QRS_NEXT_CUT()
PTP {E1 28616.968,E2 28616.968}
PTP {X 0,Y 607.867,A -85,B 0,C 180,E1 28616.968,E2 28616.968,E3 0,E4 0,E5 0,E6 0}
QRS_SPEED_INIT()
LIN {X 0,Y 607.867,Z 1084,A -85,B 0,C 180,E1 28616.968,E2 28616.968,E3 0,E4 0,E5 0,E6 0} C_VEL
LIN {X 0,Y 607.867,Z 590.149,A -85,B 0,C 180,E1 28616.968,E2 28616.968} C_VEL
LIN {X 0,Y 607.867,Z 582.07,A -85,B 0,C 180,E1 28616.968,E2 28616.968} C_VEL
LIN {X 0,Y 607.876,Z 580.07,A -85,B 0,C 180,E1 28616.78,E2 28616.78} C_VEL
LIN {X 0,Y 607.89,Z 580.076,A -85,B 0,C 180,E1 28613.483,E2 28613.483} C_VEL
LIN {X 0,Y 607.884,Z 580.069,A -85,B 0,C 180,E1 28610.437,E2 28610.437} C_VEL
LIN {X 0,Y 607.889,Z 580.074,A -85,B 0,C 180,E1 28607.17,E2 28607.17} C_VEL
LIN {X 0,Y 607.897,Z 580.069,A -85,B 0,C 180,E1 28604.057,E2 28604.057} C_VEL
LIN {X 0,Y 607.881,Z 580.073,A -85,B 0,C 180,E1 28600.758,E2 28600.758} C_VEL
LIN {X 0,Y 607.908,Z 580.069,A -85,B 0,C 180,E1 28597.67,E2 28597.67} C_VEL
LIN {X 0,Y 607.882,Z 580.073,A -85,B 0,C 180,E1 28594.472,E2 28594.472} C_VEL
LIN {X 0,Y 607.917,Z 580.068,A -85,B 0,C 180,E1 28591.405,E2 28591.405} C_VEL
LIN {X 0,Y 607.88,Z 580.072,A -85,B 0,C 180,E1 28588.13,E2 28588.13} C_VEL
LIN {X 0,Y 607.913,Z 580.071,A -85,B 0,C 180,E1 28584.993,E2 28584.993} C_VEL
LIN {X 0,Y 607.881,Z 580.072,A -85,B 0,C 180,E1 28581.834,E2 28581.834} C_VEL
LIN {X 0,Y 607.911,Z 580.072,A -85,B 0,C 180,E1 28578.734,E2 28578.734} C_VEL
LIN {X 0,Y 607.907,Z 580.227,A -85,B 0,C 180,E1 28576.36,E2 28576.36} C_VEL
LIN {X 0,Y 607.894,Z 606.241,A -85,B 0,C 180,E1 28573.564,E2 28573.564} C_VEL
LIN {X 0,Y 607.911,Z 636.019,A -85,B 0,C 180,E1 28570.459,E2 28570.459} C_VEL
LIN {X 0,Y 607.889,Z 666.862,A -85,B 0,C 180,E1 28567.309,E2 28567.309} C_VEL
LIN {X 0,Y 607.91,Z 698.053,A -85,B 0,C 180,E1 28564.176,E2 28564.176} C_VEL
LIN {X 0,Y 607.909,Z 709.953,A -85,B 0,C 180,E1 28563.027,E2 28563.027} C_VEL
LIN {X 0,Y 607.905,Z 821.643,A -85,B 0,C 180,E1 28561.66,E2 28561.66} C_VEL
LIN {X 0,Y 607.917,Z 836.088,A -85,B 0,C 180,E1 28561.314,E2 28561.314} C_VEL
LIN {X 0,Y 607.919,Z 850.913,A -85,B 0,C 180,E1 28560.764,E2 28560.764} C_VEL
LIN {X 0,Y 607.91,Z 863.899,A -85,B 0,C 180,E1 28560.101,E2 28560.101} C_VEL
LIN {X 0,Y 607.919,Z 876.772,A -85,B 0,C 180,E1 28559.241,E2 28559.241} C_VEL
LIN {X 0,Y 607.919,Z 886.967,A -85,B 0,C 180,E1 28558.366,E2 28558.366} C_VEL
LIN {X 0,Y 607.917,Z 896.549,A -85,B 0,C 180,E1 28557.357,E2 28557.357} C_VEL
LIN {X 0,Y 607.917,Z 905.81,A -85,B 0,C 180,E1 28556.1,E2 28556.1} C_VEL
LIN {X 0,Y 607.915,Z 913.073,A -85,B 0,C 180,E1 28554.783,E2 28554.783} C_VEL
LIN {X 0,Y 607.916,Z 918.363,A -85,B 0,C 180,E1 28553.455,E2 28553.455} C_VEL
LIN {X 0,Y 607.917,Z 922.064,A -85,B 0,C 180,E1 28552.024,E2 28552.024} C_VEL
LIN {X 0,Y 607.916,Z 923.86,A -85,B 0,C 180,E1 28550.507,E2 28550.507} C_VEL
LIN {X 0,Y 607.917,Z 923.652,A -85,B 0,C 180,E1 28549.105,E2 28549.105} C_VEL
LIN {X 0,Y 607.915,Z 921.709,A -85,B 0,C 180,E1 28547.715,E2 28547.715} C_VEL
LIN {X 0,Y 607.914,Z 917.979,A -85,B 0,C 180,E1 28546.335,E2 28546.335} C_VEL
LIN {X 0,Y 607.919,Z 912.759,A -85,B 0,C 180,E1 28545.062,E2 28545.062} C_VEL
LIN {X 0,Y 607.918,Z 905.726,A -85,B 0,C 180,E1 28543.797,E2 28543.797} C_VEL
LIN {X 0,Y 607.919,Z 896.434,A -85,B 0,C 180,E1 28542.539,E2 28542.539} C_VEL
LIN {X 0,Y 607.917,Z 886.306,A -85,B 0,C 180,E1 28541.479,E2 28541.479} C_VEL
LIN {X 0,Y 607.916,Z 873.406,A -85,B 0,C 180,E1 28540.423,E2 28540.423} C_VEL
LIN {X 0,Y 607.898,Z 861.256,A -85,B 0,C 180,E1 28539.658,E2 28539.658} C_VEL
LIN {X 0,Y 607.918,Z 847.253,A -85,B 0,C 180,E1 28538.989,E2 28538.989} C_VEL
LIN {X 0,Y 607.919,Z 833.117,A -85,B 0,C 180,E1 28538.512,E2 28538.512} C_VEL
LIN {X 0,Y 607.905,Z 818.973,A -85,B 0,C 180,E1 28538.203,E2 28538.203} C_VEL
LIN {X 0,Y 607.918,Z 709.961,A -85,B 0,C 180,E1 28536.884,E2 28536.884} C_VEL
LIN {X 0,Y 607.915,Z 682.218,A -85,B 0,C 180,E1 28534.15,E2 28534.15} C_VEL
LIN {X 0,Y 607.91,Z 650.544,A -85,B 0,C 180,E1 28530.942,E2 28530.942} C_VEL
LIN {X 0,Y 607.909,Z 619.504,A -85,B 0,C 180,E1 28527.738,E2 28527.738} C_VEL
LIN {X 0,Y 607.919,Z 589.094,A -85,B 0,C 180,E1 28524.526,E2 28524.526} C_VEL
LIN {X 0,Y 607.905,Z 580.175,A -85,B 0,C 180,E1 28523.531,E2 28523.531} C_VEL
LIN {X 0,Y 607.898,Z 580.068,A -85,B 0,C 180,E1 28520.342,E2 28520.342} C_VEL
LIN {X 0,Y 607.902,Z 580.075,A -85,B 0,C 180,E1 28517.171,E2 28517.171} C_VEL
LIN {X 0,Y 607.895,Z 580.068,A -85,B 0,C 180,E1 28514.057,E2 28514.057} C_VEL
LIN {X 0,Y 607.903,Z 580.074,A -85,B 0,C 180,E1 28510.894,E2 28510.894} C_VEL
LIN {X 0,Y 607.892,Z 580.069,A -85,B 0,C 180,E1 28507.771,E2 28507.771} C_VEL
LIN {X 0,Y 607.904,Z 580.073,A -85,B 0,C 180,E1 28504.578,E2 28504.578} C_VEL
LIN {X 0,Y 607.888,Z 580.07,A -85,B 0,C 180,E1 28501.442,E2 28501.442} C_VEL
LIN {X 0,Y 607.906,Z 580.073,A -85,B 0,C 180,E1 28498.353,E2 28498.353} C_VEL
LIN {X 0,Y 607.886,Z 580.07,A -85,B 0,C 180,E1 28495.162,E2 28495.162} C_VEL
LIN {X 0,Y 607.905,Z 580.073,A -85,B 0,C 180,E1 28492.037,E2 28492.037} C_VEL
LIN {X 0,Y 607.886,Z 580.07,A -85,B 0,C 180,E1 28488.983,E2 28488.983} C_VEL
LIN {X 0,Y 607.906,Z 580.073,A -85,B 0,C 180,E1 28485.817,E2 28485.817} C_VEL
LIN {X 0,Y 607.882,Z 580.07,A -85,B 0,C 180,E1 28482.662,E2 28482.662} C_VEL
LIN {X 0,Y 607.908,Z 580.073,A -85,B 0,C 180,E1 28479.533,E2 28479.533} C_VEL
LIN {X 0,Y 607.88,Z 580.071,A -85,B 0,C 180,E1 28476.426,E2 28476.426} C_VEL
LIN {X 0,Y 607.912,Z 580.073,A -85,B 0,C 180,E1 28473.322,E2 28473.322} C_VEL
LIN {X 0,Y 607.879,Z 580.07,A -85,B 0,C 180,E1 28470.22,E2 28470.22} C_VEL
LIN {X 0,Y 607.914,Z 580.073,A -85,B 0,C 180,E1 28467.103,E2 28467.103} C_VEL
LIN {X 0,Y 607.877,Z 580.07,A -85,B 0,C 180,E1 28463.971,E2 28463.971} C_VEL
LIN {X 0,Y 607.916,Z 580.075,A -85,B 0,C 180,E1 28460.898,E2 28460.898} C_VEL
LIN {X 0,Y 607.876,Z 580.07,A -85,B 0,C 180,E1 28457.716,E2 28457.716} C_VEL
LIN {X 0,Y 607.917,Z 580.075,A -85,B 0,C 180,E1 28454.672,E2 28454.672} C_VEL
LIN {X 0,Y 607.875,Z 580.071,A -85,B 0,C 180,E1 28451.48,E2 28451.48} C_VEL
LIN {X 0,Y 607.918,Z 580.073,A -85,B 0,C 180,E1 28448.322,E2 28448.322} C_VEL
LIN {X 0,Y 607.871,Z 580.071,A -85,B 0,C 180,E1 28445.191,E2 28445.191} C_VEL
LIN {X 0,Y 607.917,Z 580.073,A -85,B 0,C 180,E1 28442.074,E2 28442.074} C_VEL
LIN {X 0,Y 607.868,Z 580.071,A -85,B 0,C 180,E1 28438.963,E2 28438.963} C_VEL
LIN {X 0,Y 607.918,Z 580.074,A -85,B 0,C 180,E1 28435.85,E2 28435.85} C_VEL
LIN {X 0,Y 607.866,Z 580.071,A -85,B 0,C 180,E1 28432.686,E2 28432.686} C_VEL
LIN {X 0,Y 607.919,Z 580.074,A -85,B 0,C 180,E1 28429.577,E2 28429.577} C_VEL
LIN {X 0,Y 607.864,Z 580.072,A -85,B 0,C 180,E1 28426.441,E2 28426.441} C_VEL
LIN {X 0,Y 607.918,Z 580.075,A -85,B 0,C 180,E1 28423.371,E2 28423.371} C_VEL
LIN {X 0,Y 607.863,Z 580.072,A -85,B 0,C 180,E1 28420.194,E2 28420.194} C_VEL
LIN {X 0,Y 607.914,Z 580.077,A -85,B 0,C 180,E1 28417.16,E2 28417.16} C_VEL
LIN {X 0,Y 607.867,Z 580.071,A -85,B 0,C 180,E1 28414.053,E2 28414.053} C_VEL
LIN {X 0,Y 607.913,Z 580.078,A -85,B 0,C 180,E1 28410.975,E2 28410.975} C_VEL
LIN {X 0,Y 607.864,Z 580.072,A -85,B 0,C 180,E1 28407.796,E2 28407.796} C_VEL
LIN {X 0,Y 607.906,Z 580.078,A -85,B 0,C 180,E1 28404.738,E2 28404.738} C_VEL
LIN {X 0,Y 607.862,Z 580.072,A -85,B 0,C 180,E1 28401.555,E2 28401.555} C_VEL
LIN {X 0,Y 607.894,Z 580.077,A -85,B 0,C 180,E1 28398.593,E2 28398.593} C_VEL
LIN {X 0,Y 607.867,Z 580.071,A -85,B 0,C 180,E1 28395.384,E2 28395.384} C_VEL
LIN {X 0,Y 607.886,Z 580.077,A -85,B 0,C 180,E1 28392.394,E2 28392.394} C_VEL
LIN {X 0,Y 607.869,Z 580.072,A -85,B 0,C 180,E1 28389.171,E2 28389.171} C_VEL
LIN {X 0,Y 607.869,Z 580.076,A -85,B 0,C 180,E1 28386.295,E2 28386.295} C_VEL
LIN {X 0,Y 607.889,Z 580.07,A -85,B 0,C 180,E1 28383.099,E2 28383.099} C_VEL
LIN {X 0,Y 607.865,Z 580.075,A -85,B 0,C 180,E1 28380.094,E2 28380.094} C_VEL
LIN {X 0,Y 607.896,Z 580.312,A -85,B 0,C 180,E1 28379.784,E2 28379.784} C_VEL
LIN {X 0,Y 607.918,Z 589.008,A -85,B 0,C 180,E1 28379.15,E2 28379.15} C_VEL
LIN {X 0,Y 607.866,Z 632.567,A -85,B 0,C 180,E1 28376.209,E2 28376.209} C_VEL
LIN {X 0,Y 607.91,Z 678.154,A -85,B 0,C 180,E1 28373.205,E2 28373.205} C_VEL
LIN {X 0,Y 607.897,Z 691.997,A -85,B 0,C 180,E1 28372.331,E2 28372.331} C_VEL
LIN {X 0,Y 607.914,Z 901.305,A -85,B 0,C 180,E1 28369.705,E2 28369.705} C_VEL
LIN {X 0,Y 607.901,Z 919.582,A -85,B 0,C 180,E1 28369.305,E2 28369.305} C_VEL
LIN {X 0,Y 607.918,Z 938.403,A -85,B 0,C 180,E1 28368.707,E2 28368.707} C_VEL
LIN {X 0,Y 607.886,Z 956.055,A -85,B 0,C 180,E1 28367.963,E2 28367.963} C_VEL
LIN {X 0,Y 607.919,Z 972.787,A -85,B 0,C 180,E1 28367.073,E2 28367.073} C_VEL
LIN {X 0,Y 607.916,Z 988.639,A -85,B 0,C 180,E1 28366.041,E2 28366.041} C_VEL
LIN {X 0,Y 607.918,Z 1003.56,A -85,B 0,C 180,E1 28364.867,E2 28364.867} C_VEL
LIN {X 0,Y 607.918,Z 1017.218,A -85,B 0,C 180,E1 28363.582,E2 28363.582} C_VEL
LIN {X 0,Y 607.916,Z 1029.905,A -85,B 0,C 180,E1 28362.153,E2 28362.153} C_VEL
LIN {X 0,Y 607.915,Z 1041.223,A -85,B 0,C 180,E1 28360.615,E2 28360.615} C_VEL
LIN {X 0,Y 607.918,Z 1050.988,A -85,B 0,C 180,E1 28358.989,E2 28358.989} C_VEL
LIN {X 0,Y 607.909,Z 1058.863,A -85,B 0,C 180,E1 28357.35,E2 28357.35} C_VEL
LIN {X 0,Y 607.906,Z 1065.107,A -85,B 0,C 180,E1 28355.664,E2 28355.664} C_VEL
LIN {X 0,Y 607.916,Z 1069.872,A -85,B 0,C 180,E1 28353.867,E2 28353.867} C_VEL
LIN {X 0,Y 607.916,Z 1072.787,A -85,B 0,C 180,E1 28352.074,E2 28352.074} C_VEL
LIN {X 0,Y 607.907,Z 1073.94,A -85,B 0,C 180,E1 28350.283,E2 28350.283} C_VEL
LIN {X 0,Y 607.915,Z 1073.348,A -85,B 0,C 180,E1 28348.492,E2 28348.492} C_VEL
LIN {X 0,Y 607.908,Z 1071.005,A -85,B 0,C 180,E1 28346.7,E2 28346.7} C_VEL
LIN {X 0,Y 607.905,Z 1067.096,A -85,B 0,C 180,E1 28344.999,E2 28344.999} C_VEL
LIN {X 0,Y 607.914,Z 1061.467,A -85,B 0,C 180,E1 28343.294,E2 28343.294} C_VEL
LIN {X 0,Y 607.918,Z 1054.423,A -85,B 0,C 180,E1 28341.678,E2 28341.678} C_VEL
LIN {X 0,Y 607.91,Z 1045.509,A -85,B 0,C 180,E1 28340.055,E2 28340.055} C_VEL
LIN {X 0,Y 607.919,Z 1035.145,A -85,B 0,C 180,E1 28338.521,E2 28338.521} C_VEL
LIN {X 0,Y 607.914,Z 1023.346,A -85,B 0,C 180,E1 28337.075,E2 28337.075} C_VEL
LIN {X 0,Y 607.915,Z 1010.089,A -85,B 0,C 180,E1 28335.717,E2 28335.717} C_VEL
LIN {X 0,Y 607.917,Z 995.234,A -85,B 0,C 180,E1 28334.449,E2 28334.449} C_VEL
LIN {X 0,Y 607.918,Z 979.217,A -85,B 0,C 180,E1 28333.321,E2 28333.321} C_VEL
LIN {X 0,Y 607.895,Z 963.025,A -85,B 0,C 180,E1 28332.384,E2 28332.384} C_VEL
LIN {X 0,Y 607.907,Z 946.062,A -85,B 0,C 180,E1 28331.591,E2 28331.591} C_VEL
LIN {X 0,Y 607.905,Z 927.374,A -85,B 0,C 180,E1 28330.92,E2 28330.92} C_VEL
LIN {X 0,Y 607.905,Z 909.317,A -85,B 0,C 180,E1 28330.449,E2 28330.449} C_VEL
LIN {X 0,Y 607.919,Z 889.788,A -85,B 0,C 180,E1 28330.128,E2 28330.128} C_VEL
LIN {X 0,Y 607.896,Z 691.355,A -85,B 0,C 180,E1 28327.646,E2 28327.646} C_VEL
LIN {X 0,Y 607.914,Z 645.175,A -85,B 0,C 180,E1 28324.631,E2 28324.631} C_VEL
LIN {X 0,Y 607.917,Z 598.704,A -85,B 0,C 180,E1 28321.512,E2 28321.512} C_VEL
LIN {X 0,Y 607.898,Z 580.397,A -85,B 0,C 180,E1 28320.232,E2 28320.232} C_VEL
LIN {X 0,Y 607.853,Z 580.073,A -85,B 0,C 180,E1 28319.342,E2 28319.342} C_VEL
LIN {X 0,Y 607.909,Z 580.078,A -85,B 0,C 180,E1 28316.16,E2 28316.16} C_VEL
LIN {X 0,Y 607.847,Z 580.075,A -85,B 0,C 180,E1 28313.22,E2 28313.22} C_VEL
LIN {X 0,Y 607.918,Z 580.073,A -85,B 0,C 180,E1 28310.182,E2 28310.182} C_VEL
LIN {X 0,Y 607.848,Z 580.075,A -85,B 0,C 180,E1 28307.192,E2 28307.192} C_VEL
LIN {X 0,Y 607.919,Z 580.069,A -85,B 0,C 180,E1 28304.184,E2 28304.184} C_VEL
LIN {X 0,Y 607.851,Z 580.076,A -85,B 0,C 180,E1 28301.02,E2 28301.02} C_VEL
LIN {X 0,Y 607.909,Z 580.069,A -85,B 0,C 180,E1 28298.016,E2 28298.016} C_VEL
LIN {X 0,Y 607.855,Z 580.076,A -85,B 0,C 180,E1 28294.835,E2 28294.835} C_VEL
LIN {X 0,Y 607.897,Z 580.069,A -85,B 0,C 180,E1 28291.869,E2 28291.869} C_VEL
LIN {X 0,Y 607.862,Z 580.076,A -85,B 0,C 180,E1 28288.705,E2 28288.705} C_VEL
LIN {X 0,Y 607.886,Z 580.07,A -85,B 0,C 180,E1 28285.736,E2 28285.736} C_VEL
LIN {X 0,Y 607.869,Z 580.077,A -85,B 0,C 180,E1 28282.535,E2 28282.535} C_VEL
LIN {X 0,Y 607.876,Z 580.07,A -85,B 0,C 180,E1 28279.606,E2 28279.606} C_VEL
LIN {X 0,Y 607.873,Z 580.077,A -85,B 0,C 180,E1 28276.336,E2 28276.336} C_VEL
LIN {X 0,Y 607.882,Z 580.07,A -85,B 0,C 180,E1 28273.313,E2 28273.313} C_VEL
LIN {X 0,Y 607.875,Z 580.076,A -85,B 0,C 180,E1 28270.041,E2 28270.041} C_VEL
LIN {X 0,Y 607.891,Z 580.069,A -85,B 0,C 180,E1 28266.991,E2 28266.991} C_VEL
LIN {X 0,Y 607.875,Z 580.076,A -85,B 0,C 180,E1 28263.772,E2 28263.772} C_VEL
LIN {X 0,Y 607.889,Z 580.069,A -85,B 0,C 180,E1 28260.754,E2 28260.754} C_VEL
LIN {X 0,Y 607.881,Z 580.075,A -85,B 0,C 180,E1 28257.549,E2 28257.549} C_VEL
LIN {X 0,Y 607.876,Z 580.07,A -85,B 0,C 180,E1 28256.78,E2 28256.78} C_VEL
LIN {X 0,Y 606.932,Z 580.196,A -85,B 0,C 180,E1 28256.054,E2 28256.054} C_VEL
LIN {X 0,Y 600.424,Z 581.012,A -85,B 0,C 180,E1 28253.964,E2 28253.964} C_VEL
LIN {X 0,Y 599.952,Z 581.065,A -85,B 0,C 180,E1 28253.487,E2 28253.487} C_VEL
LIN {X 0,Y 599.948,Z 581.058,A -85,B 0,C 180,E1 28250.406,E2 28250.406} C_VEL
LIN {X 0,Y 599.944,Z 581.063,A -85,B 0,C 180,E1 28247.096,E2 28247.096} C_VEL
LIN {X 0,Y 599.971,Z 581.057,A -85,B 0,C 180,E1 28243.94,E2 28243.94} C_VEL
LIN {X 0,Y 599.94,Z 581.062,A -85,B 0,C 180,E1 28240.732,E2 28240.732} C_VEL
LIN {X 0,Y 599.97,Z 581.058,A -85,B 0,C 180,E1 28237.656,E2 28237.656} C_VEL
LIN {X 0,Y 599.941,Z 581.062,A -85,B 0,C 180,E1 28234.427,E2 28234.427} C_VEL
LIN {X 0,Y 599.974,Z 581.059,A -85,B 0,C 180,E1 28231.317,E2 28231.317} C_VEL
LIN {X 0,Y 599.941,Z 581.061,A -85,B 0,C 180,E1 28228.108,E2 28228.108} C_VEL
LIN {X 0,Y 599.975,Z 581.059,A -85,B 0,C 180,E1 28225.021,E2 28225.021} C_VEL
LIN {X 0,Y 599.942,Z 581.061,A -85,B 0,C 180,E1 28221.807,E2 28221.807} C_VEL
LIN {X 0,Y 599.972,Z 581.062,A -85,B 0,C 180,E1 28218.704,E2 28218.704} C_VEL
LIN {X 0,Y 600.003,Z 581.296,A -85,B 0,C 180,E1 28216.611,E2 28216.611} C_VEL
LIN {X 0,Y 600.305,Z 585.322,A -85,B 0,C 180,E1 28216.141,E2 28216.141} C_VEL
LIN {X 0,Y 600.216,Z 615.031,A -85,B 0,C 180,E1 28212.947,E2 28212.947} C_VEL
LIN {X 0,Y 600.138,Z 645.674,A -85,B 0,C 180,E1 28209.729,E2 28209.729} C_VEL
LIN {X 0,Y 600.077,Z 677.028,A -85,B 0,C 180,E1 28206.501,E2 28206.501} C_VEL
LIN {X 0,Y 600.029,Z 709.286,A -85,B 0,C 180,E1 28203.246,E2 28203.246} C_VEL
LIN {X 0,Y 600.113,Z 712.197,A -85,B 0,C 180,E1 28203.155,E2 28203.155} C_VEL
LIN {X 0,Y 600.068,Z 821.391,A -85,B 0,C 180,E1 28201.819,E2 28201.819} C_VEL
LIN {X 0,Y 600.062,Z 836.233,A -85,B 0,C 180,E1 28201.461,E2 28201.461} C_VEL
LIN {X 0,Y 600.039,Z 850.43,A -85,B 0,C 180,E1 28200.929,E2 28200.929} C_VEL
LIN {X 0,Y 600.003,Z 863.74,A -85,B 0,C 180,E1 28200.246,E2 28200.246} C_VEL
LIN {X 0,Y 599.985,Z 876.43,A -85,B 0,C 180,E1 28199.392,E2 28199.392} C_VEL
LIN {X 0,Y 599.962,Z 887.649,A -85,B 0,C 180,E1 28198.411,E2 28198.411} C_VEL
LIN {X 0,Y 599.942,Z 897.114,A -85,B 0,C 180,E1 28197.386,E2 28197.386} C_VEL
LIN {X 0,Y 599.931,Z 905.633,A -85,B 0,C 180,E1 28196.21,E2 28196.21} C_VEL
LIN {X 0,Y 599.923,Z 912.634,A -85,B 0,C 180,E1 28194.939,E2 28194.939} C_VEL
LIN {X 0,Y 599.92,Z 917.785,A -85,B 0,C 180,E1 28193.682,E2 28193.682} C_VEL
LIN {X 0,Y 599.917,Z 921.699,A -85,B 0,C 180,E1 28192.23,E2 28192.23} C_VEL
LIN {X 0,Y 599.918,Z 923.597,A -85,B 0,C 180,E1 28190.895,E2 28190.895} C_VEL
LIN {X 0,Y 599.915,Z 923.894,A -85,B 0,C 180,E1 28189.471,E2 28189.471} C_VEL
LIN {X 0,Y 599.917,Z 922.396,A -85,B 0,C 180,E1 28188.059,E2 28188.059} C_VEL
LIN {X 0,Y 599.917,Z 919.149,A -85,B 0,C 180,E1 28186.658,E2 28186.658} C_VEL
LIN {X 0,Y 599.919,Z 914.02,A -85,B 0,C 180,E1 28185.268,E2 28185.268} C_VEL
LIN {X 0,Y 599.93,Z 907.355,A -85,B 0,C 180,E1 28183.984,E2 28183.984} C_VEL
LIN {X 0,Y 599.936,Z 899.376,A -85,B 0,C 180,E1 28182.806,E2 28182.806} C_VEL
LIN {X 0,Y 599.958,Z 889.975,A -85,B 0,C 180,E1 28181.731,E2 28181.731} C_VEL
LIN {X 0,Y 599.977,Z 880.494,A -85,B 0,C 180,E1 28180.854,E2 28180.854} C_VEL
LIN {X 0,Y 599.976,Z 869.55,A -85,B 0,C 180,E1 28180.029,E2 28180.029} C_VEL
LIN {X 0,Y 600.023,Z 857.202,A -85,B 0,C 180,E1 28179.302,E2 28179.302} C_VEL
LIN {X 0,Y 600.05,Z 842.832,A -85,B 0,C 180,E1 28178.673,E2 28178.673} C_VEL
LIN {X 0,Y 600.074,Z 828.414,A -85,B 0,C 180,E1 28178.238,E2 28178.238} C_VEL
LIN {X 0,Y 600.07,Z 813.09,A -85,B 0,C 180,E1 28177.966,E2 28177.966} C_VEL
LIN {X 0,Y 600.055,Z 710.005,A -85,B 0,C 180,E1 28176.711,E2 28176.711} C_VEL
LIN {X 0,Y 600.033,Z 688.618,A -85,B 0,C 180,E1 28174.588,E2 28174.588} C_VEL
LIN {X 0,Y 600.092,Z 657.766,A -85,B 0,C 180,E1 28171.432,E2 28171.432} C_VEL
LIN {X 0,Y 600.176,Z 627.511,A -85,B 0,C 180,E1 28168.281,E2 28168.281} C_VEL
LIN {X 0,Y 600.269,Z 597.858,A -85,B 0,C 180,E1 28165.127,E2 28165.127} C_VEL
LIN {X 0,Y 600.134,Z 582.003,A -85,B 0,C 180,E1 28163.399,E2 28163.399} C_VEL
LIN {X 0,Y 599.961,Z 581.085,A -85,B 0,C 180,E1 28163.204,E2 28163.204} C_VEL
LIN {X 0,Y 599.954,Z 581.061,A -85,B 0,C 180,E1 28160.045,E2 28160.045} C_VEL
LIN {X 0,Y 599.96,Z 581.06,A -85,B 0,C 180,E1 28156.9,E2 28156.9} C_VEL
LIN {X 0,Y 599.952,Z 581.061,A -85,B 0,C 180,E1 28153.741,E2 28153.741} C_VEL
LIN {X 0,Y 599.963,Z 581.058,A -85,B 0,C 180,E1 28150.53,E2 28150.53} C_VEL
LIN {X 0,Y 599.954,Z 581.062,A -85,B 0,C 180,E1 28147.357,E2 28147.357} C_VEL
LIN {X 0,Y 599.971,Z 581.056,A -85,B 0,C 180,E1 28144.111,E2 28144.111} C_VEL
LIN {X 0,Y 599.973,Z 581.065,A -85,B 0,C 180,E1 28140.772,E2 28140.772} C_VEL
LIN {X 0,Y 599.954,Z 581.056,A -85,B 0,C 180,E1 28137.432,E2 28137.432} C_VEL
LIN {X 0,Y 599.97,Z 581.063,A -85,B 0,C 180,E1 28134.252,E2 28134.252} C_VEL
LIN {X 0,Y 599.948,Z 581.058,A -85,B 0,C 180,E1 28131.075,E2 28131.075} C_VEL
LIN {X 0,Y 599.97,Z 581.062,A -85,B 0,C 180,E1 28127.937,E2 28127.937} C_VEL
LIN {X 0,Y 599.945,Z 581.059,A -85,B 0,C 180,E1 28124.767,E2 28124.767} C_VEL
LIN {X 0,Y 599.971,Z 581.061,A -85,B 0,C 180,E1 28121.678,E2 28121.678} C_VEL
LIN {X 0,Y 599.944,Z 581.059,A -85,B 0,C 180,E1 28118.558,E2 28118.558} C_VEL
LIN {X 0,Y 599.97,Z 581.062,A -85,B 0,C 180,E1 28115.419,E2 28115.419} C_VEL
LIN {X 0,Y 599.943,Z 581.058,A -85,B 0,C 180,E1 28112.331,E2 28112.331} C_VEL
LIN {X 0,Y 599.975,Z 581.062,A -85,B 0,C 180,E1 28109.161,E2 28109.161} C_VEL
LIN {X 0,Y 599.938,Z 581.058,A -85,B 0,C 180,E1 28105.997,E2 28105.997} C_VEL
LIN {X 0,Y 599.974,Z 581.062,A -85,B 0,C 180,E1 28102.849,E2 28102.849} C_VEL
LIN {X 0,Y 599.937,Z 581.06,A -85,B 0,C 180,E1 28099.775,E2 28099.775} C_VEL
LIN {X 0,Y 599.974,Z 581.061,A -85,B 0,C 180,E1 28096.615,E2 28096.615} C_VEL
LIN {X 0,Y 599.934,Z 581.06,A -85,B 0,C 180,E1 28093.493,E2 28093.493} C_VEL
LIN {X 0,Y 599.977,Z 581.06,A -85,B 0,C 180,E1 28090.369,E2 28090.369} C_VEL
LIN {X 0,Y 599.934,Z 581.059,A -85,B 0,C 180,E1 28087.277,E2 28087.277} C_VEL
LIN {X 0,Y 599.977,Z 581.062,A -85,B 0,C 180,E1 28084.11,E2 28084.11} C_VEL
LIN {X 0,Y 599.927,Z 581.06,A -85,B 0,C 180,E1 28080.955,E2 28080.955} C_VEL
LIN {X 0,Y 599.978,Z 581.063,A -85,B 0,C 180,E1 28077.899,E2 28077.899} C_VEL
LIN {X 0,Y 599.927,Z 581.061,A -85,B 0,C 180,E1 28074.741,E2 28074.741} C_VEL
LIN {X 0,Y 599.979,Z 581.063,A -85,B 0,C 180,E1 28071.664,E2 28071.664} C_VEL
LIN {X 0,Y 599.926,Z 581.061,A -85,B 0,C 180,E1 28068.519,E2 28068.519} C_VEL
LIN {X 0,Y 599.98,Z 581.063,A -85,B 0,C 180,E1 28065.426,E2 28065.426} C_VEL
LIN {X 0,Y 599.928,Z 581.061,A -85,B 0,C 180,E1 28062.343,E2 28062.343} C_VEL
LIN {X 0,Y 599.978,Z 581.064,A -85,B 0,C 180,E1 28059.214,E2 28059.214} C_VEL
LIN {X 0,Y 599.927,Z 581.061,A -85,B 0,C 180,E1 28056.11,E2 28056.11} C_VEL
LIN {X 0,Y 599.977,Z 581.065,A -85,B 0,C 180,E1 28053.045,E2 28053.045} C_VEL
LIN {X 0,Y 599.926,Z 581.06,A -85,B 0,C 180,E1 28049.882,E2 28049.882} C_VEL
LIN {X 0,Y 599.966,Z 581.066,A -85,B 0,C 180,E1 28046.865,E2 28046.865} C_VEL
LIN {X 0,Y 599.932,Z 581.06,A -85,B 0,C 180,E1 28043.726,E2 28043.726} C_VEL
LIN {X 0,Y 599.951,Z 581.065,A -85,B 0,C 180,E1 28040.706,E2 28040.706} C_VEL
LIN {X 0,Y 599.925,Z 581.061,A -85,B 0,C 180,E1 28037.417,E2 28037.417} C_VEL
LIN {X 0,Y 599.963,Z 581.066,A -85,B 0,C 180,E1 28034.362,E2 28034.362} C_VEL
LIN {X 0,Y 599.92,Z 581.062,A -85,B 0,C 180,E1 28031.121,E2 28031.121} C_VEL
LIN {X 0,Y 599.966,Z 581.066,A -85,B 0,C 180,E1 28028.07,E2 28028.07} C_VEL
LIN {X 0,Y 599.919,Z 581.063,A -85,B 0,C 180,E1 28024.867,E2 28024.867} C_VEL
LIN {X 0,Y 599.955,Z 581.066,A -85,B 0,C 180,E1 28021.891,E2 28021.891} C_VEL
LIN {X 0,Y 599.958,Z 581.314,A -85,B 0,C 180,E1 28020.144,E2 28020.144} C_VEL
LIN {X 0,Y 600.654,Z 584.52,A -85,B 0,C 180,E1 28019.85,E2 28019.85} C_VEL
LIN {X 0,Y 600.468,Z 627.841,A -85,B 0,C 180,E1 28016.878,E2 28016.878} C_VEL
LIN {X 0,Y 600.389,Z 672.736,A -85,B 0,C 180,E1 28013.871,E2 28013.871} C_VEL
LIN {X 0,Y 600.409,Z 692.171,A -85,B 0,C 180,E1 28012.621,E2 28012.621} C_VEL
LIN {X 0,Y 600.373,Z 901.305,A -85,B 0,C 180,E1 28009.963,E2 28009.963} C_VEL
LIN {X 0,Y 600.32,Z 920.323,A -85,B 0,C 180,E1 28009.538,E2 28009.538} C_VEL
LIN {X 0,Y 600.29,Z 938.402,A -85,B 0,C 180,E1 28008.954,E2 28008.954} C_VEL
LIN {X 0,Y 600.204,Z 956.053,A -85,B 0,C 180,E1 28008.201,E2 28008.201} C_VEL
LIN {X 0,Y 600.18,Z 972.703,A -85,B 0,C 180,E1 28007.305,E2 28007.305} C_VEL
LIN {X 0,Y 600.122,Z 988.638,A -85,B 0,C 180,E1 28006.255,E2 28006.255} C_VEL
LIN {X 0,Y 600.069,Z 1003.561,A -85,B 0,C 180,E1 28005.066,E2 28005.066} C_VEL
LIN {X 0,Y 600.02,Z 1017.017,A -85,B 0,C 180,E1 28003.786,E2 28003.786} C_VEL
LIN {X 0,Y 599.983,Z 1029.906,A -85,B 0,C 180,E1 28002.317,E2 28002.317} C_VEL
LIN {X 0,Y 599.956,Z 1041.224,A -85,B 0,C 180,E1 28000.758,E2 28000.758} C_VEL
LIN {X 0,Y 599.934,Z 1050.989,A -85,B 0,C 180,E1 27999.11,E2 27999.11} C_VEL
LIN {X 0,Y 599.92,Z 1059.042,A -85,B 0,C 180,E1 27997.406,E2 27997.406} C_VEL
LIN {X 0,Y 599.91,Z 1065.409,A -85,B 0,C 180,E1 27995.643,E2 27995.643} C_VEL
LIN {X 0,Y 599.916,Z 1069.873,A -85,B 0,C 180,E1 27993.918,E2 27993.918} C_VEL
LIN {X 0,Y 599.917,Z 1072.787,A -85,B 0,C 180,E1 27992.102,E2 27992.102} C_VEL
LIN {X 0,Y 599.907,Z 1073.94,A -85,B 0,C 180,E1 27990.287,E2 27990.287} C_VEL
LIN {X 0,Y 599.915,Z 1073.348,A -85,B 0,C 180,E1 27988.472,E2 27988.472} C_VEL
LIN {X 0,Y 599.907,Z 1071.005,A -85,B 0,C 180,E1 27986.656,E2 27986.656} C_VEL
LIN {X 0,Y 599.908,Z 1067.097,A -85,B 0,C 180,E1 27984.932,E2 27984.932} C_VEL
LIN {X 0,Y 599.92,Z 1061.468,A -85,B 0,C 180,E1 27983.204,E2 27983.204} C_VEL
LIN {X 0,Y 599.931,Z 1054.423,A -85,B 0,C 180,E1 27981.567,E2 27981.567} C_VEL
LIN {X 0,Y 599.942,Z 1045.51,A -85,B 0,C 180,E1 27979.922,E2 27979.922} C_VEL
LIN {X 0,Y 599.969,Z 1035.146,A -85,B 0,C 180,E1 27978.367,E2 27978.367} C_VEL
LIN {X 0,Y 600,Z 1023.346,A -85,B 0,C 180,E1 27976.901,E2 27976.901} C_VEL
LIN {X 0,Y 600.047,Z 1009.759,A -85,B 0,C 180,E1 27975.494,E2 27975.494} C_VEL
LIN {X 0,Y 600.103,Z 995.233,A -85,B 0,C 180,E1 27974.242,E2 27974.242} C_VEL
LIN {X 0,Y 600.165,Z 979.22,A -85,B 0,C 180,E1 27973.099,E2 27973.099} C_VEL
LIN {X 0,Y 600.195,Z 962.033,A -85,B 0,C 180,E1 27972.1,E2 27972.1} C_VEL
LIN {X 0,Y 600.277,Z 944.644,A -85,B 0,C 180,E1 27971.293,E2 27971.293} C_VEL
LIN {X 0,Y 600.315,Z 926.513,A -85,B 0,C 180,E1 27970.644,E2 27970.644} C_VEL
LIN {X 0,Y 600.358,Z 908.143,A -85,B 0,C 180,E1 27970.17,E2 27970.17} C_VEL
LIN {X 0,Y 600.395,Z 888.268,A -85,B 0,C 180,E1 27969.85,E2 27969.85} C_VEL
LIN {X 0,Y 600.37,Z 691.85,A -85,B 0,C 180,E1 27967.371,E2 27967.371} C_VEL
LIN {X 0,Y 600.463,Z 645.962,A -85,B 0,C 180,E1 27964.346,E2 27964.346} C_VEL
LIN {X 0,Y 600.604,Z 599.492,A -85,B 0,C 180,E1 27961.187,E2 27961.187} C_VEL
LIN {X 0,Y 600.562,Z 583.327,A -85,B 0,C 180,E1 27960.062,E2 27960.062} C_VEL
LIN {X 0,Y 599.949,Z 581.259,A -85,B 0,C 180,E1 27959.842,E2 27959.842} C_VEL
LIN {X 0,Y 599.943,Z 581.06,A -85,B 0,C 180,E1 27956.96,E2 27956.96} C_VEL
LIN {X 0,Y 599.93,Z 581.066,A -85,B 0,C 180,E1 27953.726,E2 27953.726} C_VEL
LIN {X 0,Y 599.933,Z 581.061,A -85,B 0,C 180,E1 27950.803,E2 27950.803} C_VEL
LIN {X 0,Y 599.936,Z 581.066,A -85,B 0,C 180,E1 27947.548,E2 27947.548} C_VEL
LIN {X 0,Y 599.934,Z 581.06,A -85,B 0,C 180,E1 27944.559,E2 27944.559} C_VEL
LIN {X 0,Y 599.931,Z 581.066,A -85,B 0,C 180,E1 27941.267,E2 27941.267} C_VEL
LIN {X 0,Y 599.939,Z 581.059,A -85,B 0,C 180,E1 27938.282,E2 27938.282} C_VEL
LIN {X 0,Y 599.927,Z 581.065,A -85,B 0,C 180,E1 27934.982,E2 27934.982} C_VEL
LIN {X 0,Y 599.947,Z 581.059,A -85,B 0,C 180,E1 27931.974,E2 27931.974} C_VEL
LIN {X 0,Y 599.929,Z 581.065,A -85,B 0,C 180,E1 27928.759,E2 27928.759} C_VEL
LIN {X 0,Y 599.942,Z 581.06,A -85,B 0,C 180,E1 27925.784,E2 27925.784} C_VEL
LIN {X 0,Y 599.931,Z 581.066,A -85,B 0,C 180,E1 27922.54,E2 27922.54} C_VEL
LIN {X 0,Y 599.94,Z 581.059,A -85,B 0,C 180,E1 27919.572,E2 27919.572} C_VEL
LIN {X 0,Y 599.929,Z 581.065,A -85,B 0,C 180,E1 27916.26,E2 27916.26} C_VEL
LIN {X 0,Y 599.947,Z 581.058,A -85,B 0,C 180,E1 27913.274,E2 27913.274} C_VEL
LIN {X 0,Y 599.932,Z 581.063,A -85,B 0,C 180,E1 27909.981,E2 27909.981} C_VEL
LIN {X 0,Y 599.963,Z 581.058,A -85,B 0,C 180,E1 27906.891,E2 27906.891} C_VEL
LIN {X 0,Y 599.928,Z 581.064,A -85,B 0,C 180,E1 27903.631,E2 27903.631} C_VEL
LIN {X 0,Y 599.972,Z 581.057,A -85,B 0,C 180,E1 27900.573,E2 27900.573} C_VEL
LIN {X 0,Y 599.934,Z 581.063,A -85,B 0,C 180,E1 27897.421,E2 27897.421} C_VEL
LIN {X 0,Y 599.97,Z 581.057,A -85,B 0,C 180,E1 27894.357,E2 27894.357} C_VEL
LIN {X 0,Y 599.952,Z 581.065,A -85,B 0,C 180,E1 27893.487,E2 27893.487} C_VEL
LIN {X 0,Y 598.92,Z 581.19,A -85,B 0,C 180,E1 27892.751,E2 27892.751} C_VEL
LIN {X 0,Y 592.538,Z 581.981,A -85,B 0,C 180,E1 27890.687,E2 27890.687} C_VEL
LIN {X 0,Y 592.031,Z 582.045,A -85,B 0,C 180,E1 27890.15,E2 27890.15} C_VEL
LIN {X 0,Y 591.996,Z 582.05,A -85,B 0,C 180,E1 27886.919,E2 27886.919} C_VEL
LIN {X 0,Y 592.04,Z 582.047,A -85,B 0,C 180,E1 27883.82,E2 27883.82} C_VEL
LIN {X 0,Y 591.996,Z 582.05,A -85,B 0,C 180,E1 27880.565,E2 27880.565} C_VEL
LIN {X 0,Y 592.035,Z 582.049,A -85,B 0,C 180,E1 27877.457,E2 27877.457} C_VEL
LIN {X 0,Y 591.999,Z 582.05,A -85,B 0,C 180,E1 27874.274,E2 27874.274} C_VEL
LIN {X 0,Y 592.031,Z 582.051,A -85,B 0,C 180,E1 27871.117,E2 27871.117} C_VEL
LIN {X 0,Y 591.999,Z 582.05,A -85,B 0,C 180,E1 27867.972,E2 27867.972} C_VEL
LIN {X 0,Y 592.034,Z 582.052,A -85,B 0,C 180,E1 27864.826,E2 27864.826} C_VEL
LIN {X 0,Y 592.001,Z 582.05,A -85,B 0,C 180,E1 27861.695,E2 27861.695} C_VEL
LIN {X 0,Y 592.034,Z 582.053,A -85,B 0,C 180,E1 27858.545,E2 27858.545} C_VEL
LIN {X 0,Y 592.074,Z 582.327,A -85,B 0,C 180,E1 27856.881,E2 27856.881} C_VEL
LIN {X 0,Y 592.702,Z 586.499,A -85,B 0,C 180,E1 27856.372,E2 27856.372} C_VEL
LIN {X 0,Y 592.524,Z 616.438,A -85,B 0,C 180,E1 27853.112,E2 27853.112} C_VEL
LIN {X 0,Y 592.364,Z 647.333,A -85,B 0,C 180,E1 27849.825,E2 27849.825} C_VEL
LIN {X 0,Y 592.236,Z 678.433,A -85,B 0,C 180,E1 27846.581,E2 27846.581} C_VEL
LIN {X 0,Y 592.145,Z 709.618,A -85,B 0,C 180,E1 27843.399,E2 27843.399} C_VEL
LIN {X 0,Y 592.323,Z 714.866,A -85,B 0,C 180,E1 27843.3,E2 27843.3} C_VEL
LIN {X 0,Y 592.235,Z 821.487,A -85,B 0,C 180,E1 27841.977,E2 27841.977} C_VEL
LIN {X 0,Y 592.215,Z 835.505,A -85,B 0,C 180,E1 27841.637,E2 27841.637} C_VEL
LIN {X 0,Y 592.164,Z 849.69,A -85,B 0,C 180,E1 27841.11,E2 27841.11} C_VEL
LIN {X 0,Y 592.106,Z 862.876,A -85,B 0,C 180,E1 27840.437,E2 27840.437} C_VEL
LIN {X 0,Y 592.053,Z 876.075,A -85,B 0,C 180,E1 27839.546,E2 27839.546} C_VEL
LIN {X 0,Y 592.006,Z 887.393,A -85,B 0,C 180,E1 27838.553,E2 27838.553} C_VEL
LIN {X 0,Y 591.972,Z 896.748,A -85,B 0,C 180,E1 27837.533,E2 27837.533} C_VEL
LIN {X 0,Y 591.945,Z 905.951,A -85,B 0,C 180,E1 27836.244,E2 27836.244} C_VEL
LIN {X 0,Y 591.927,Z 913.27,A -85,B 0,C 180,E1 27834.872,E2 27834.872} C_VEL
LIN {X 0,Y 591.92,Z 918.538,A -85,B 0,C 180,E1 27833.494,E2 27833.494} C_VEL
LIN {X 0,Y 591.918,Z 921.975,A -85,B 0,C 180,E1 27832.129,E2 27832.129} C_VEL
LIN {X 0,Y 591.916,Z 923.781,A -85,B 0,C 180,E1 27830.639,E2 27830.639} C_VEL
LIN {X 0,Y 591.916,Z 923.747,A -85,B 0,C 180,E1 27829.22,E2 27829.22} C_VEL
LIN {X 0,Y 591.917,Z 922.015,A -85,B 0,C 180,E1 27827.803,E2 27827.803} C_VEL
LIN {X 0,Y 591.918,Z 918.392,A -85,B 0,C 180,E1 27826.37,E2 27826.37} C_VEL
LIN {X 0,Y 591.929,Z 913.459,A -85,B 0,C 180,E1 27825.078,E2 27825.078} C_VEL
LIN {X 0,Y 591.943,Z 906.024,A -85,B 0,C 180,E1 27823.679,E2 27823.679} C_VEL
LIN {X 0,Y 591.968,Z 897.606,A -85,B 0,C 180,E1 27822.486,E2 27822.486} C_VEL
LIN {X 0,Y 592.003,Z 888.76,A -85,B 0,C 180,E1 27821.496,E2 27821.496} C_VEL
LIN {X 0,Y 592.04,Z 879.052,A -85,B 0,C 180,E1 27820.608,E2 27820.608} C_VEL
LIN {X 0,Y 592.071,Z 866.962,A -85,B 0,C 180,E1 27819.722,E2 27819.722} C_VEL
LIN {X 0,Y 592.155,Z 852.718,A -85,B 0,C 180,E1 27818.937,E2 27818.937} C_VEL
LIN {X 0,Y 592.202,Z 839.325,A -85,B 0,C 180,E1 27818.398,E2 27818.398} C_VEL
LIN {X 0,Y 592.239,Z 824.513,A -85,B 0,C 180,E1 27817.991,E2 27817.991} C_VEL
LIN {X 0,Y 592.246,Z 802.911,A -85,B 0,C 180,E1 27817.681,E2 27817.681} C_VEL
LIN {X 0,Y 592.206,Z 710.405,A -85,B 0,C 180,E1 27816.544,E2 27816.544} C_VEL
LIN {X 0,Y 592.124,Z 708.342,A -85,B 0,C 180,E1 27816.399,E2 27816.399} C_VEL
LIN {X 0,Y 592.232,Z 676.194,A -85,B 0,C 180,E1 27813.097,E2 27813.097} C_VEL
LIN {X 0,Y 592.379,Z 644.687,A -85,B 0,C 180,E1 27809.806,E2 27809.806} C_VEL
LIN {X 0,Y 592.535,Z 613.827,A -85,B 0,C 180,E1 27806.517,E2 27806.517} C_VEL
LIN {X 0,Y 592.695,Z 584.935,A -85,B 0,C 180,E1 27803.364,E2 27803.364} C_VEL
LIN {X 0,Y 592.036,Z 582.127,A -85,B 0,C 180,E1 27802.967,E2 27802.967} C_VEL
LIN {X 0,Y 592.029,Z 582.055,A -85,B 0,C 180,E1 27799.687,E2 27799.687} C_VEL
LIN {X 0,Y 592.029,Z 582.045,A -85,B 0,C 180,E1 27796.323,E2 27796.323} C_VEL
LIN {X 0,Y 592.029,Z 582.053,A -85,B 0,C 180,E1 27793.012,E2 27793.012} C_VEL
LIN {X 0,Y 592.015,Z 582.047,A -85,B 0,C 180,E1 27789.846,E2 27789.846} C_VEL
LIN {X 0,Y 592.027,Z 582.048,A -85,B 0,C 180,E1 27786.721,E2 27786.721} C_VEL
LIN {X 0,Y 592.011,Z 582.048,A -85,B 0,C 180,E1 27783.52,E2 27783.52} C_VEL
LIN {X 0,Y 592.026,Z 582.047,A -85,B 0,C 180,E1 27780.34,E2 27780.34} C_VEL
LIN {X 0,Y 592.008,Z 582.047,A -85,B 0,C 180,E1 27777.17,E2 27777.17} C_VEL
LIN {X 0,Y 592.026,Z 582.049,A -85,B 0,C 180,E1 27773.996,E2 27773.996} C_VEL
LIN {X 0,Y 592.007,Z 582.049,A -85,B 0,C 180,E1 27770.825,E2 27770.825} C_VEL
LIN {X 0,Y 592.029,Z 582.046,A -85,B 0,C 180,E1 27767.634,E2 27767.634} C_VEL
LIN {X 0,Y 592.006,Z 582.051,A -85,B 0,C 180,E1 27764.5,E2 27764.5} C_VEL
LIN {X 0,Y 592.033,Z 582.044,A -85,B 0,C 180,E1 27761.275,E2 27761.275} C_VEL
LIN {X 0,Y 592.007,Z 582.052,A -85,B 0,C 180,E1 27758.089,E2 27758.089} C_VEL
LIN {X 0,Y 592.033,Z 582.043,A -85,B 0,C 180,E1 27754.809,E2 27754.809} C_VEL
LIN {X 0,Y 592.037,Z 582.055,A -85,B 0,C 180,E1 27751.457,E2 27751.457} C_VEL
LIN {X 0,Y 592.003,Z 582.048,A -85,B 0,C 180,E1 27748.16,E2 27748.16} C_VEL
LIN {X 0,Y 592.034,Z 582.05,A -85,B 0,C 180,E1 27744.975,E2 27744.975} C_VEL
LIN {X 0,Y 591.997,Z 582.049,A -85,B 0,C 180,E1 27741.813,E2 27741.813} C_VEL
LIN {X 0,Y 592.036,Z 582.047,A -85,B 0,C 180,E1 27738.657,E2 27738.657} C_VEL
LIN {X 0,Y 591.992,Z 582.049,A -85,B 0,C 180,E1 27735.478,E2 27735.478} C_VEL
LIN {X 0,Y 592.036,Z 582.049,A -85,B 0,C 180,E1 27732.385,E2 27732.385} C_VEL
LIN {X 0,Y 591.991,Z 582.048,A -85,B 0,C 180,E1 27729.233,E2 27729.233} C_VEL
LIN {X 0,Y 592.037,Z 582.049,A -85,B 0,C 180,E1 27726.108,E2 27726.108} C_VEL
LIN {X 0,Y 591.989,Z 582.05,A -85,B 0,C 180,E1 27723.001,E2 27723.001} C_VEL
LIN {X 0,Y 592.039,Z 582.049,A -85,B 0,C 180,E1 27719.903,E2 27719.903} C_VEL
LIN {X 0,Y 591.988,Z 582.05,A -85,B 0,C 180,E1 27716.805,E2 27716.805} C_VEL
LIN {X 0,Y 592.04,Z 582.048,A -85,B 0,C 180,E1 27713.698,E2 27713.698} C_VEL
LIN {X 0,Y 591.986,Z 582.05,A -85,B 0,C 180,E1 27710.533,E2 27710.533} C_VEL
LIN {X 0,Y 592.04,Z 582.05,A -85,B 0,C 180,E1 27707.417,E2 27707.417} C_VEL
LIN {X 0,Y 591.984,Z 582.05,A -85,B 0,C 180,E1 27704.31,E2 27704.31} C_VEL
LIN {X 0,Y 592.04,Z 582.05,A -85,B 0,C 180,E1 27701.182,E2 27701.182} C_VEL
LIN {X 0,Y 591.979,Z 582.051,A -85,B 0,C 180,E1 27698.014,E2 27698.014} C_VEL
LIN {X 0,Y 592.041,Z 582.05,A -85,B 0,C 180,E1 27694.919,E2 27694.919} C_VEL
LIN {X 0,Y 591.977,Z 582.052,A -85,B 0,C 180,E1 27691.776,E2 27691.776} C_VEL
LIN {X 0,Y 592.04,Z 582.052,A -85,B 0,C 180,E1 27688.711,E2 27688.711} C_VEL
LIN {X 0,Y 591.976,Z 582.051,A -85,B 0,C 180,E1 27685.541,E2 27685.541} C_VEL
LIN {X 0,Y 592.042,Z 582.051,A -85,B 0,C 180,E1 27682.435,E2 27682.435} C_VEL
LIN {X 0,Y 591.976,Z 582.052,A -85,B 0,C 180,E1 27679.31,E2 27679.31} C_VEL
LIN {X 0,Y 592.04,Z 582.054,A -85,B 0,C 180,E1 27676.289,E2 27676.289} C_VEL
LIN {X 0,Y 591.978,Z 582.051,A -85,B 0,C 180,E1 27673.143,E2 27673.143} C_VEL
LIN {X 0,Y 592.039,Z 582.055,A -85,B 0,C 180,E1 27670.05,E2 27670.05} C_VEL
LIN {X 0,Y 591.981,Z 582.051,A -85,B 0,C 180,E1 27666.963,E2 27666.963} C_VEL
LIN {X 0,Y 592.017,Z 582.057,A -85,B 0,C 180,E1 27663.978,E2 27663.978} C_VEL
LIN {X 0,Y 591.979,Z 582.05,A -85,B 0,C 180,E1 27660.716,E2 27660.716} C_VEL
LIN {X 0,Y 592.057,Z 582.577,A -85,B 0,C 180,E1 27660.477,E2 27660.477} C_VEL
LIN {X 0,Y 593.397,Z 586.883,A -85,B 0,C 180,E1 27660.085,E2 27660.085} C_VEL
LIN {X 0,Y 593.075,Z 630.204,A -85,B 0,C 180,E1 27657.078,E2 27657.078} C_VEL
LIN {X 0,Y 592.875,Z 674.312,A -85,B 0,C 180,E1 27654.087,E2 27654.087} C_VEL
LIN {X 0,Y 592.861,Z 692.208,A -85,B 0,C 180,E1 27652.925,E2 27652.925} C_VEL
LIN {X 0,Y 593.098,Z 707.228,A -85,B 0,C 180,E1 27652.719,E2 27652.719} C_VEL
LIN {X 0,Y 592.848,Z 901.305,A -85,B 0,C 180,E1 27650.227,E2 27650.227} C_VEL
LIN {X 0,Y 592.758,Z 920.298,A -85,B 0,C 180,E1 27649.798,E2 27649.798} C_VEL
LIN {X 0,Y 592.681,Z 938.4,A -85,B 0,C 180,E1 27649.206,E2 27649.206} C_VEL
LIN {X 0,Y 592.541,Z 956.051,A -85,B 0,C 180,E1 27648.445,E2 27648.445} C_VEL
LIN {X 0,Y 592.459,Z 972.696,A -85,B 0,C 180,E1 27647.538,E2 27647.538} C_VEL
LIN {X 0,Y 592.342,Z 988.636,A -85,B 0,C 180,E1 27646.474,E2 27646.474} C_VEL
LIN {X 0,Y 592.23,Z 1003.561,A -85,B 0,C 180,E1 27645.271,E2 27645.271} C_VEL
LIN {X 0,Y 592.131,Z 1017.017,A -85,B 0,C 180,E1 27643.973,E2 27643.973} C_VEL
LIN {X 0,Y 592.059,Z 1029.411,A -85,B 0,C 180,E1 27642.548,E2 27642.548} C_VEL
LIN {X 0,Y 591.999,Z 1040.586,A -85,B 0,C 180,E1 27641.003,E2 27641.003} C_VEL
LIN {X 0,Y 591.954,Z 1050.473,A -85,B 0,C 180,E1 27639.332,E2 27639.332} C_VEL
LIN {X 0,Y 591.935,Z 1058.772,A -85,B 0,C 180,E1 27637.571,E2 27637.571} C_VEL
LIN {X 0,Y 591.913,Z 1065.262,A -85,B 0,C 180,E1 27635.767,E2 27635.767} C_VEL
LIN {X 0,Y 591.916,Z 1069.873,A -85,B 0,C 180,E1 27633.972,E2 27633.972} C_VEL
LIN {X 0,Y 591.917,Z 1072.788,A -85,B 0,C 180,E1 27632.13,E2 27632.13} C_VEL
LIN {X 0,Y 591.907,Z 1073.94,A -85,B 0,C 180,E1 27630.291,E2 27630.291} C_VEL
LIN {X 0,Y 591.915,Z 1073.349,A -85,B 0,C 180,E1 27628.451,E2 27628.451} C_VEL
LIN {X 0,Y 591.907,Z 1071.006,A -85,B 0,C 180,E1 27626.611,E2 27626.611} C_VEL
LIN {X 0,Y 591.912,Z 1067.098,A -85,B 0,C 180,E1 27624.864,E2 27624.864} C_VEL
LIN {X 0,Y 591.928,Z 1061.468,A -85,B 0,C 180,E1 27623.112,E2 27623.112} C_VEL
LIN {X 0,Y 591.944,Z 1054.424,A -85,B 0,C 180,E1 27621.452,E2 27621.452} C_VEL
LIN {X 0,Y 591.976,Z 1045.511,A -85,B 0,C 180,E1 27619.785,E2 27619.785} C_VEL
LIN {X 0,Y 592.024,Z 1035.146,A -85,B 0,C 180,E1 27618.208,E2 27618.208} C_VEL
LIN {X 0,Y 592.093,Z 1023.347,A -85,B 0,C 180,E1 27616.723,E2 27616.723} C_VEL
LIN {X 0,Y 592.193,Z 1009.581,A -85,B 0,C 180,E1 27615.28,E2 27615.28} C_VEL
LIN {X 0,Y 592.305,Z 994.595,A -85,B 0,C 180,E1 27613.978,E2 27613.978} C_VEL
LIN {X 0,Y 592.421,Z 978.419,A -85,B 0,C 180,E1 27612.821,E2 27612.821} C_VEL
LIN {X 0,Y 592.508,Z 962.034,A -85,B 0,C 180,E1 27611.86,E2 27611.86} C_VEL
LIN {X 0,Y 592.649,Z 945.096,A -85,B 0,C 180,E1 27611.061,E2 27611.061} C_VEL
LIN {X 0,Y 592.737,Z 926.731,A -85,B 0,C 180,E1 27610.392,E2 27610.392} C_VEL
LIN {X 0,Y 592.821,Z 908.306,A -85,B 0,C 180,E1 27609.911,E2 27609.911} C_VEL
LIN {X 0,Y 592.883,Z 888.526,A -85,B 0,C 180,E1 27609.586,E2 27609.586} C_VEL
LIN {X 0,Y 592.946,Z 692.817,A -85,B 0,C 180,E1 27607.09,E2 27607.09} C_VEL
LIN {X 0,Y 592.78,Z 690.071,A -85,B 0,C 180,E1 27606.963,E2 27606.963} C_VEL
LIN {X 0,Y 593.035,Z 642.443,A -85,B 0,C 180,E1 27603.76,E2 27603.76} C_VEL
LIN {X 0,Y 593.329,Z 597.129,A -85,B 0,C 180,E1 27600.634,E2 27600.634} C_VEL
LIN {X 0,Y 593.22,Z 586.004,A -85,B 0,C 180,E1 27599.843,E2 27599.843} C_VEL
LIN {X 0,Y 592.003,Z 582.265,A -85,B 0,C 180,E1 27599.47,E2 27599.47} C_VEL
LIN {X 0,Y 592.039,Z 582.049,A -85,B 0,C 180,E1 27596.478,E2 27596.478} C_VEL
LIN {X 0,Y 591.972,Z 582.054,A -85,B 0,C 180,E1 27593.4,E2 27593.4} C_VEL
LIN {X 0,Y 592.041,Z 582.049,A -85,B 0,C 180,E1 27590.329,E2 27590.329} C_VEL
LIN {X 0,Y 591.973,Z 582.054,A -85,B 0,C 180,E1 27587.235,E2 27587.235} C_VEL
LIN {X 0,Y 592.037,Z 582.047,A -85,B 0,C 180,E1 27584.226,E2 27584.226} C_VEL
LIN {X 0,Y 591.977,Z 582.054,A -85,B 0,C 180,E1 27581.073,E2 27581.073} C_VEL
LIN {X 0,Y 592.027,Z 582.046,A -85,B 0,C 180,E1 27578.056,E2 27578.056} C_VEL
LIN {X 0,Y 591.979,Z 582.054,A -85,B 0,C 180,E1 27574.829,E2 27574.829} C_VEL
LIN {X 0,Y 592.026,Z 582.047,A -85,B 0,C 180,E1 27571.798,E2 27571.798} C_VEL
LIN {X 0,Y 591.981,Z 582.054,A -85,B 0,C 180,E1 27568.664,E2 27568.664} C_VEL
LIN {X 0,Y 592.022,Z 582.047,A -85,B 0,C 180,E1 27565.617,E2 27565.617} C_VEL
LIN {X 0,Y 591.982,Z 582.055,A -85,B 0,C 180,E1 27562.44,E2 27562.44} C_VEL
LIN {X 0,Y 592.017,Z 582.047,A -85,B 0,C 180,E1 27559.433,E2 27559.433} C_VEL
LIN {X 0,Y 591.986,Z 582.054,A -85,B 0,C 180,E1 27556.181,E2 27556.181} C_VEL
LIN {X 0,Y 592.018,Z 582.047,A -85,B 0,C 180,E1 27553.179,E2 27553.179} C_VEL
LIN {X 0,Y 591.99,Z 582.051,A -85,B 0,C 180,E1 27549.92,E2 27549.92} C_VEL
LIN {X 0,Y 592.031,Z 582.047,A -85,B 0,C 180,E1 27546.789,E2 27546.789} C_VEL
LIN {X 0,Y 591.988,Z 582.052,A -85,B 0,C 180,E1 27543.583,E2 27543.583} C_VEL
LIN {X 0,Y 592.039,Z 582.046,A -85,B 0,C 180,E1 27540.484,E2 27540.484} C_VEL
LIN {X 0,Y 591.99,Z 582.052,A -85,B 0,C 180,E1 27537.289,E2 27537.289} C_VEL
LIN {X 0,Y 592.036,Z 582.046,A -85,B 0,C 180,E1 27534.184,E2 27534.184} C_VEL
LIN {X 0,Y 591.991,Z 582.049,A -85,B 0,C 180,E1 27530.963,E2 27530.963} C_VEL
LIN {X 0,Y 592.031,Z 582.045,A -85,B 0,C 180,E1 27530.15,E2 27530.15} C_VEL
LIN {X 0,Y 591.06,Z 582.174,A -85,B 0,C 180,E1 27529.404,E2 27529.404} C_VEL
LIN {X 0,Y 584.594,Z 582.978,A -85,B 0,C 180,E1 27527.313,E2 27527.313} C_VEL
LIN {X 0,Y 584.053,Z 583.038,A -85,B 0,C 180,E1 27526.768,E2 27526.768} C_VEL
LIN {X 0,Y 584.096,Z 583.04,A -85,B 0,C 180,E1 27523.593,E2 27523.593} C_VEL
LIN {X 0,Y 584.056,Z 583.039,A -85,B 0,C 180,E1 27520.395,E2 27520.395} C_VEL
LIN {X 0,Y 584.097,Z 583.042,A -85,B 0,C 180,E1 27517.24,E2 27517.24} C_VEL
LIN {X 0,Y 584.058,Z 583.038,A -85,B 0,C 180,E1 27514.116,E2 27514.116} C_VEL
LIN {X 0,Y 584.097,Z 583.044,A -85,B 0,C 180,E1 27510.912,E2 27510.912} C_VEL
LIN {X 0,Y 584.064,Z 583.038,A -85,B 0,C 180,E1 27507.716,E2 27507.716} C_VEL
LIN {X 0,Y 584.096,Z 583.043,A -85,B 0,C 180,E1 27504.401,E2 27504.401} C_VEL
LIN {X 0,Y 584.092,Z 583.037,A -85,B 0,C 180,E1 27501.079,E2 27501.079} C_VEL
LIN {X 0,Y 584.076,Z 583.044,A -85,B 0,C 180,E1 27497.837,E2 27497.837} C_VEL
LIN {X 0,Y 584.099,Z 583.234,A -85,B 0,C 180,E1 27497.188,E2 27497.188} C_VEL
LIN {X 0,Y 585.104,Z 587.998,A -85,B 0,C 180,E1 27496.574,E2 27496.574} C_VEL
LIN {X 0,Y 584.834,Z 617.844,A -85,B 0,C 180,E1 27493.28,E2 27493.28} C_VEL
LIN {X 0,Y 584.598,Z 648.43,A -85,B 0,C 180,E1 27489.983,E2 27489.983} C_VEL
LIN {X 0,Y 584.397,Z 679.838,A -85,B 0,C 180,E1 27486.663,E2 27486.663} C_VEL
LIN {X 0,Y 584.271,Z 709.893,A -85,B 0,C 180,E1 27483.568,E2 27483.568} C_VEL
LIN {X 0,Y 584.536,Z 716.942,A -85,B 0,C 180,E1 27483.455,E2 27483.455} C_VEL
LIN {X 0,Y 584.407,Z 821.486,A -85,B 0,C 180,E1 27482.14,E2 27482.14} C_VEL
LIN {X 0,Y 584.368,Z 836.249,A -85,B 0,C 180,E1 27481.774,E2 27481.774} C_VEL
LIN {X 0,Y 584.29,Z 851.054,A -85,B 0,C 180,E1 27481.201,E2 27481.201} C_VEL
LIN {X 0,Y 584.2,Z 864.063,A -85,B 0,C 180,E1 27480.508,E2 27480.508} C_VEL
LIN {X 0,Y 584.123,Z 876.442,A -85,B 0,C 180,E1 27479.649,E2 27479.649} C_VEL
LIN {X 0,Y 584.052,Z 887.681,A -85,B 0,C 180,E1 27478.642,E2 27478.642} C_VEL
LIN {X 0,Y 583.999,Z 897.125,A -85,B 0,C 180,E1 27477.589,E2 27477.589} C_VEL
LIN {X 0,Y 583.958,Z 905.981,A -85,B 0,C 180,E1 27476.325,E2 27476.325} C_VEL
LIN {X 0,Y 583.933,Z 913.401,A -85,B 0,C 180,E1 27474.912,E2 27474.912} C_VEL
LIN {X 0,Y 583.921,Z 918.625,A -85,B 0,C 180,E1 27473.514,E2 27473.514} C_VEL
LIN {X 0,Y 583.919,Z 922.039,A -85,B 0,C 180,E1 27472.123,E2 27472.123} C_VEL
LIN {X 0,Y 583.916,Z 923.848,A -85,B 0,C 180,E1 27470.55,E2 27470.55} C_VEL
LIN {X 0,Y 583.917,Z 923.642,A -85,B 0,C 180,E1 27469.054,E2 27469.054} C_VEL
LIN {X 0,Y 583.916,Z 921.753,A -85,B 0,C 180,E1 27467.643,E2 27467.643} C_VEL
LIN {X 0,Y 583.922,Z 917.813,A -85,B 0,C 180,E1 27466.134,E2 27466.134} C_VEL
LIN {X 0,Y 583.938,Z 911.83,A -85,B 0,C 180,E1 27464.661,E2 27464.661} C_VEL
LIN {X 0,Y 583.957,Z 904.576,A -85,B 0,C 180,E1 27463.365,E2 27463.365} C_VEL
LIN {X 0,Y 584.009,Z 895.774,A -85,B 0,C 180,E1 27462.152,E2 27462.152} C_VEL
LIN {X 0,Y 584.082,Z 884.515,A -85,B 0,C 180,E1 27460.954,E2 27460.954} C_VEL
LIN {X 0,Y 584.137,Z 872.387,A -85,B 0,C 180,E1 27459.955,E2 27459.955} C_VEL
LIN {X 0,Y 584.223,Z 859.874,A -85,B 0,C 180,E1 27459.158,E2 27459.158} C_VEL
LIN {X 0,Y 584.317,Z 846.571,A -85,B 0,C 180,E1 27458.512,E2 27458.512} C_VEL
LIN {X 0,Y 584.389,Z 831.026,A -85,B 0,C 180,E1 27457.984,E2 27457.984} C_VEL
LIN {X 0,Y 584.419,Z 815.755,A -85,B 0,C 180,E1 27457.676,E2 27457.676} C_VEL
LIN {X 0,Y 584.34,Z 710.602,A -85,B 0,C 180,E1 27456.364,E2 27456.364} C_VEL
LIN {X 0,Y 584.237,Z 708.607,A -85,B 0,C 180,E1 27456.239,E2 27456.239} C_VEL
LIN {X 0,Y 584.412,Z 675.999,A -85,B 0,C 180,E1 27452.844,E2 27452.844} C_VEL
LIN {X 0,Y 584.621,Z 644.525,A -85,B 0,C 180,E1 27449.51,E2 27449.51} C_VEL
LIN {X 0,Y 584.852,Z 614.598,A -85,B 0,C 180,E1 27446.275,E2 27446.275} C_VEL
LIN {X 0,Y 585.1,Z 587.262,A -85,B 0,C 180,E1 27443.253,E2 27443.253} C_VEL
LIN {X 0,Y 584.115,Z 583.159,A -85,B 0,C 180,E1 27442.698,E2 27442.698} C_VEL
LIN {X 0,Y 584.09,Z 583.044,A -85,B 0,C 180,E1 27439.346,E2 27439.346} C_VEL
LIN {X 0,Y 584.078,Z 583.037,A -85,B 0,C 180,E1 27436.08,E2 27436.08} C_VEL
LIN {X 0,Y 584.086,Z 583.04,A -85,B 0,C 180,E1 27432.876,E2 27432.876} C_VEL
LIN {X 0,Y 584.073,Z 583.037,A -85,B 0,C 180,E1 27429.665,E2 27429.665} C_VEL
LIN {X 0,Y 584.086,Z 583.032,A -85,B 0,C 180,E1 27426.493,E2 27426.493} C_VEL
LIN {X 0,Y 584.072,Z 583.039,A -85,B 0,C 180,E1 27423.33,E2 27423.33} C_VEL
LIN {X 0,Y 584.088,Z 583.031,A -85,B 0,C 180,E1 27420.122,E2 27420.122} C_VEL
LIN {X 0,Y 584.074,Z 583.038,A -85,B 0,C 180,E1 27416.901,E2 27416.901} C_VEL
LIN {X 0,Y 584.096,Z 583.033,A -85,B 0,C 180,E1 27413.558,E2 27413.558} C_VEL
LIN {X 0,Y 584.099,Z 583.043,A -85,B 0,C 180,E1 27410.192,E2 27410.192} C_VEL
LIN {X 0,Y 584.07,Z 583.034,A -85,B 0,C 180,E1 27406.918,E2 27406.918} C_VEL
LIN {X 0,Y 584.093,Z 583.04,A -85,B 0,C 180,E1 27403.748,E2 27403.748} C_VEL
LIN {X 0,Y 584.064,Z 583.035,A -85,B 0,C 180,E1 27400.528,E2 27400.528} C_VEL
LIN {X 0,Y 584.093,Z 583.039,A -85,B 0,C 180,E1 27397.412,E2 27397.412} C_VEL
LIN {X 0,Y 584.062,Z 583.036,A -85,B 0,C 180,E1 27394.223,E2 27394.223} C_VEL
LIN {X 0,Y 584.093,Z 583.037,A -85,B 0,C 180,E1 27391.015,E2 27391.015} C_VEL
LIN {X 0,Y 584.059,Z 583.039,A -85,B 0,C 180,E1 27387.863,E2 27387.863} C_VEL
LIN {X 0,Y 584.096,Z 583.034,A -85,B 0,C 180,E1 27384.636,E2 27384.636} C_VEL
LIN {X 0,Y 584.058,Z 583.041,A -85,B 0,C 180,E1 27381.491,E2 27381.491} C_VEL
LIN {X 0,Y 584.096,Z 583.03,A -85,B 0,C 180,E1 27378.256,E2 27378.256} C_VEL
LIN {X 0,Y 584.062,Z 583.041,A -85,B 0,C 180,E1 27375.083,E2 27375.083} C_VEL
LIN {X 0,Y 584.078,Z 583.035,A -85,B 0,C 180,E1 27371.754,E2 27371.754} C_VEL
LIN {X 0,Y 584.098,Z 583.04,A -85,B 0,C 180,E1 27368.466,E2 27368.466} C_VEL
LIN {X 0,Y 584.055,Z 583.038,A -85,B 0,C 180,E1 27365.206,E2 27365.206} C_VEL
LIN {X 0,Y 584.099,Z 583.037,A -85,B 0,C 180,E1 27362.06,E2 27362.06} C_VEL
LIN {X 0,Y 584.05,Z 583.037,A -85,B 0,C 180,E1 27358.921,E2 27358.921} C_VEL
LIN {X 0,Y 584.101,Z 583.039,A -85,B 0,C 180,E1 27355.779,E2 27355.779} C_VEL
LIN {X 0,Y 584.047,Z 583.036,A -85,B 0,C 180,E1 27352.623,E2 27352.623} C_VEL
LIN {X 0,Y 584.1,Z 583.039,A -85,B 0,C 180,E1 27349.446,E2 27349.446} C_VEL
LIN {X 0,Y 584.044,Z 583.039,A -85,B 0,C 180,E1 27346.335,E2 27346.335} C_VEL
LIN {X 0,Y 584.101,Z 583.039,A -85,B 0,C 180,E1 27343.185,E2 27343.185} C_VEL
LIN {X 0,Y 584.042,Z 583.04,A -85,B 0,C 180,E1 27340.031,E2 27340.031} C_VEL
LIN {X 0,Y 584.101,Z 583.039,A -85,B 0,C 180,E1 27336.921,E2 27336.921} C_VEL
LIN {X 0,Y 584.038,Z 583.039,A -85,B 0,C 180,E1 27333.777,E2 27333.777} C_VEL
LIN {X 0,Y 584.102,Z 583.037,A -85,B 0,C 180,E1 27330.611,E2 27330.611} C_VEL
LIN {X 0,Y 584.039,Z 583.041,A -85,B 0,C 180,E1 27327.566,E2 27327.566} C_VEL
LIN {X 0,Y 584.102,Z 583.039,A -85,B 0,C 180,E1 27324.401,E2 27324.401} C_VEL
LIN {X 0,Y 584.033,Z 583.04,A -85,B 0,C 180,E1 27321.322,E2 27321.322} C_VEL
LIN {X 0,Y 584.102,Z 583.041,A -85,B 0,C 180,E1 27318.25,E2 27318.25} C_VEL
LIN {X 0,Y 584.034,Z 583.041,A -85,B 0,C 180,E1 27315.135,E2 27315.135} C_VEL
LIN {X 0,Y 584.093,Z 583.045,A -85,B 0,C 180,E1 27312.147,E2 27312.147} C_VEL
LIN {X 0,Y 584.04,Z 583.041,A -85,B 0,C 180,E1 27308.992,E2 27308.992} C_VEL
LIN {X 0,Y 584.091,Z 583.045,A -85,B 0,C 180,E1 27305.934,E2 27305.934} C_VEL
LIN {X 0,Y 584.037,Z 583.04,A -85,B 0,C 180,E1 27302.751,E2 27302.751} C_VEL
LIN {X 0,Y 584.082,Z 583.2,A -85,B 0,C 180,E1 27300.93,E2 27300.93} C_VEL
LIN {X 0,Y 585.506,Z 587.671,A -85,B 0,C 180,E1 27300.477,E2 27300.477} C_VEL
LIN {X 0,Y 586.144,Z 589.955,A -85,B 0,C 180,E1 27300.276,E2 27300.276} C_VEL
LIN {X 0,Y 585.687,Z 632.567,A -85,B 0,C 180,E1 27297.282,E2 27297.282} C_VEL
LIN {X 0,Y 585.36,Z 676.774,A -85,B 0,C 180,E1 27294.249,E2 27294.249} C_VEL
LIN {X 0,Y 585.31,Z 692.115,A -85,B 0,C 180,E1 27293.24,E2 27293.24} C_VEL
LIN {X 0,Y 585.73,Z 697.875,A -85,B 0,C 180,E1 27293.143,E2 27293.143} C_VEL
LIN {X 0,Y 585.338,Z 901.305,A -85,B 0,C 180,E1 27290.498,E2 27290.498} C_VEL
LIN {X 0,Y 585.209,Z 920.297,A -85,B 0,C 180,E1 27290.064,E2 27290.064} C_VEL
LIN {X 0,Y 585.085,Z 938.398,A -85,B 0,C 180,E1 27289.466,E2 27289.466} C_VEL
LIN {X 0,Y 584.892,Z 956.047,A -85,B 0,C 180,E1 27288.695,E2 27288.695} C_VEL
LIN {X 0,Y 584.738,Z 973.221,A -85,B 0,C 180,E1 27287.744,E2 27287.744} C_VEL
LIN {X 0,Y 584.56,Z 989.234,A -85,B 0,C 180,E1 27286.654,E2 27286.654} C_VEL
LIN {X 0,Y 584.393,Z 1004.1,A -85,B 0,C 180,E1 27285.431,E2 27285.431} C_VEL
LIN {X 0,Y 584.241,Z 1017.943,A -85,B 0,C 180,E1 27284.065,E2 27284.065} C_VEL
LIN {X 0,Y 584.126,Z 1030.682,A -85,B 0,C 180,E1 27282.556,E2 27282.556} C_VEL
LIN {X 0,Y 584.041,Z 1041.864,A -85,B 0,C 180,E1 27280.955,E2 27280.955} C_VEL
LIN {X 0,Y 583.976,Z 1051.508,A -85,B 0,C 180,E1 27279.262,E2 27279.262} C_VEL
LIN {X 0,Y 583.942,Z 1059.402,A -85,B 0,C 180,E1 27277.521,E2 27277.521} C_VEL
LIN {X 0,Y 583.917,Z 1065.41,A -85,B 0,C 180,E1 27275.799,E2 27275.799} C_VEL
LIN {X 0,Y 583.917,Z 1069.874,A -85,B 0,C 180,E1 27274.026,E2 27274.026} C_VEL
LIN {X 0,Y 583.917,Z 1072.789,A -85,B 0,C 180,E1 27272.159,E2 27272.159} C_VEL
LIN {X 0,Y 583.907,Z 1073.94,A -85,B 0,C 180,E1 27270.295,E2 27270.295} C_VEL
LIN {X 0,Y 583.914,Z 1073.349,A -85,B 0,C 180,E1 27268.43,E2 27268.43} C_VEL
LIN {X 0,Y 583.907,Z 1071.006,A -85,B 0,C 180,E1 27266.564,E2 27266.564} C_VEL
LIN {X 0,Y 583.916,Z 1067.098,A -85,B 0,C 180,E1 27264.793,E2 27264.793} C_VEL
LIN {X 0,Y 583.934,Z 1061.468,A -85,B 0,C 180,E1 27263.017,E2 27263.017} C_VEL
LIN {X 0,Y 583.958,Z 1054.424,A -85,B 0,C 180,E1 27261.334,E2 27261.334} C_VEL
LIN {X 0,Y 584.015,Z 1045.512,A -85,B 0,C 180,E1 27259.644,E2 27259.644} C_VEL
LIN {X 0,Y 584.086,Z 1035.148,A -85,B 0,C 180,E1 27258.046,E2 27258.046} C_VEL
LIN {X 0,Y 584.194,Z 1023.348,A -85,B 0,C 180,E1 27256.54,E2 27256.54} C_VEL
LIN {X 0,Y 584.344,Z 1009.58,A -85,B 0,C 180,E1 27255.077,E2 27255.077} C_VEL
LIN {X 0,Y 584.508,Z 994.597,A -85,B 0,C 180,E1 27253.759,E2 27253.759} C_VEL
LIN {X 0,Y 584.685,Z 978.422,A -85,B 0,C 180,E1 27252.587,E2 27252.587} C_VEL
LIN {X 0,Y 584.833,Z 961.708,A -85,B 0,C 180,E1 27251.596,E2 27251.596} C_VEL
LIN {X 0,Y 585.035,Z 944.797,A -85,B 0,C 180,E1 27250.792,E2 27250.792} C_VEL
LIN {X 0,Y 585.172,Z 926.626,A -85,B 0,C 180,E1 27250.125,E2 27250.125} C_VEL
LIN {X 0,Y 585.299,Z 908.144,A -85,B 0,C 180,E1 27249.638,E2 27249.638} C_VEL
LIN {X 0,Y 585.385,Z 888.3,A -85,B 0,C 180,E1 27249.31,E2 27249.31} C_VEL
LIN {X 0,Y 585.566,Z 693.834,A -85,B 0,C 180,E1 27246.798,E2 27246.798} C_VEL
LIN {X 0,Y 585.246,Z 690.883,A -85,B 0,C 180,E1 27246.703,E2 27246.703} C_VEL
LIN {X 0,Y 585.622,Z 642.812,A -85,B 0,C 180,E1 27243.428,E2 27243.428} C_VEL
LIN {X 0,Y 586.058,Z 598.704,A -85,B 0,C 180,E1 27240.346,E2 27240.346} C_VEL
LIN {X 0,Y 586.113,Z 589.252,A -85,B 0,C 180,E1 27239.672,E2 27239.672} C_VEL
LIN {X 0,Y 584.1,Z 583.341,A -85,B 0,C 180,E1 27239.1,E2 27239.1} C_VEL
LIN {X 0,Y 584.058,Z 583.044,A -85,B 0,C 180,E1 27237.93,E2 27237.93} C_VEL
LIN {X 0,Y 584.063,Z 583.04,A -85,B 0,C 180,E1 27234.886,E2 27234.886} C_VEL
LIN {X 0,Y 584.047,Z 583.044,A -85,B 0,C 180,E1 27231.579,E2 27231.579} C_VEL
LIN {X 0,Y 584.079,Z 583.037,A -85,B 0,C 180,E1 27228.51,E2 27228.51} C_VEL
LIN {X 0,Y 584.04,Z 583.044,A -85,B 0,C 180,E1 27225.273,E2 27225.273} C_VEL
LIN {X 0,Y 584.08,Z 583.038,A -85,B 0,C 180,E1 27222.28,E2 27222.28} C_VEL
LIN {X 0,Y 584.042,Z 583.042,A -85,B 0,C 180,E1 27219.05,E2 27219.05} C_VEL
LIN {X 0,Y 584.073,Z 583.037,A -85,B 0,C 180,E1 27216.078,E2 27216.078} C_VEL
LIN {X 0,Y 584.045,Z 583.043,A -85,B 0,C 180,E1 27212.867,E2 27212.867} C_VEL
LIN {X 0,Y 584.083,Z 583.037,A -85,B 0,C 180,E1 27209.784,E2 27209.784} C_VEL
LIN {X 0,Y 584.041,Z 583.043,A -85,B 0,C 180,E1 27206.54,E2 27206.54} C_VEL
LIN {X 0,Y 584.092,Z 583.035,A -85,B 0,C 180,E1 27203.431,E2 27203.431} C_VEL
LIN {X 0,Y 584.042,Z 583.041,A -85,B 0,C 180,E1 27200.232,E2 27200.232} C_VEL
LIN {X 0,Y 584.097,Z 583.036,A -85,B 0,C 180,E1 27197.123,E2 27197.123} C_VEL
LIN {X 0,Y 584.043,Z 583.04,A -85,B 0,C 180,E1 27193.907,E2 27193.907} C_VEL
LIN {X 0,Y 584.096,Z 583.037,A -85,B 0,C 180,E1 27190.853,E2 27190.853} C_VEL
LIN {X 0,Y 584.047,Z 583.041,A -85,B 0,C 180,E1 27187.674,E2 27187.674} C_VEL
LIN {X 0,Y 584.099,Z 583.036,A -85,B 0,C 180,E1 27184.516,E2 27184.516} C_VEL
LIN {X 0,Y 584.046,Z 583.04,A -85,B 0,C 180,E1 27181.373,E2 27181.373} C_VEL
LIN {X 0,Y 584.097,Z 583.038,A -85,B 0,C 180,E1 27178.234,E2 27178.234} C_VEL
LIN {X 0,Y 584.05,Z 583.038,A -85,B 0,C 180,E1 27175.089,E2 27175.089} C_VEL
LIN {X 0,Y 584.098,Z 583.04,A -85,B 0,C 180,E1 27171.931,E2 27171.931} C_VEL
LIN {X 0,Y 584.053,Z 583.039,A -85,B 0,C 180,E1 27168.746,E2 27168.746} C_VEL
LIN {X 0,Y 584.053,Z 583.038,A -85,B 0,C 180,E1 27166.768,E2 27166.768} C_VEL
LIN {X 0,Y 583.068,Z 583.162,A -85,B 0,C 180,E1 27166.012,E2 27166.012} C_VEL
LIN {X 0,Y 576.687,Z 583.97,A -85,B 0,C 180,E1 27163.891,E2 27163.891} C_VEL
LIN {X 0,Y 576.158,Z 584.031,A -85,B 0,C 180,E1 27163.339,E2 27163.339} C_VEL
LIN {X 0,Y 576.126,Z 584.026,A -85,B 0,C 180,E1 27160.113,E2 27160.113} C_VEL
LIN {X 0,Y 576.143,Z 584.029,A -85,B 0,C 180,E1 27156.8,E2 27156.8} C_VEL
LIN {X 0,Y 576.157,Z 584.025,A -85,B 0,C 180,E1 27153.513,E2 27153.513} C_VEL
LIN {X 0,Y 576.124,Z 584.029,A -85,B 0,C 180,E1 27150.198,E2 27150.198} C_VEL
LIN {X 0,Y 576.155,Z 584.029,A -85,B 0,C 180,E1 27146.981,E2 27146.981} C_VEL
LIN {X 0,Y 576.125,Z 584.029,A -85,B 0,C 180,E1 27143.804,E2 27143.804} C_VEL
LIN {X 0,Y 576.154,Z 584.031,A -85,B 0,C 180,E1 27140.697,E2 27140.697} C_VEL
LIN {X 0,Y 576.145,Z 584.164,A -85,B 0,C 180,E1 27137.509,E2 27137.509} C_VEL
LIN {X 0,Y 577.505,Z 590.076,A -85,B 0,C 180,E1 27136.716,E2 27136.716} C_VEL
LIN {X 0,Y 577.15,Z 619.25,A -85,B 0,C 180,E1 27133.454,E2 27133.454} C_VEL
LIN {X 0,Y 576.831,Z 649.894,A -85,B 0,C 180,E1 27130.105,E2 27130.105} C_VEL
LIN {X 0,Y 576.558,Z 681.174,A -85,B 0,C 180,E1 27126.755,E2 27126.755} C_VEL
LIN {X 0,Y 576.391,Z 709.912,A -85,B 0,C 180,E1 27123.757,E2 27123.757} C_VEL
LIN {X 0,Y 576.76,Z 716.514,A -85,B 0,C 180,E1 27123.646,E2 27123.646} C_VEL
LIN {X 0,Y 576.584,Z 821.401,A -85,B 0,C 180,E1 27122.31,E2 27122.31} C_VEL
LIN {X 0,Y 576.527,Z 836.305,A -85,B 0,C 180,E1 27121.935,E2 27121.935} C_VEL
LIN {X 0,Y 576.421,Z 851.032,A -85,B 0,C 180,E1 27121.358,E2 27121.358} C_VEL
LIN {X 0,Y 576.299,Z 864.574,A -85,B 0,C 180,E1 27120.622,E2 27120.622} C_VEL
LIN {X 0,Y 576.194,Z 876.794,A -85,B 0,C 180,E1 27119.755,E2 27119.755} C_VEL
LIN {X 0,Y 576.1,Z 887.969,A -85,B 0,C 180,E1 27118.734,E2 27118.734} C_VEL
LIN {X 0,Y 576.033,Z 896.947,A -85,B 0,C 180,E1 27117.718,E2 27117.718} C_VEL
LIN {X 0,Y 575.973,Z 905.472,A -85,B 0,C 180,E1 27116.496,E2 27116.496} C_VEL
LIN {X 0,Y 575.941,Z 912.525,A -85,B 0,C 180,E1 27115.172,E2 27115.172} C_VEL
LIN {X 0,Y 575.924,Z 918.054,A -85,B 0,C 180,E1 27113.752,E2 27113.752} C_VEL
LIN {X 0,Y 575.918,Z 921.878,A -85,B 0,C 180,E1 27112.239,E2 27112.239} C_VEL
LIN {X 0,Y 575.916,Z 923.726,A -85,B 0,C 180,E1 27110.742,E2 27110.742} C_VEL
LIN {X 0,Y 575.916,Z 923.788,A -85,B 0,C 180,E1 27109.26,E2 27109.26} C_VEL
LIN {X 0,Y 575.917,Z 922.096,A -85,B 0,C 180,E1 27107.792,E2 27107.792} C_VEL
LIN {X 0,Y 575.92,Z 918.589,A -85,B 0,C 180,E1 27106.335,E2 27106.335} C_VEL
LIN {X 0,Y 575.939,Z 913.68,A -85,B 0,C 180,E1 27104.991,E2 27104.991} C_VEL
LIN {X 0,Y 575.97,Z 906.311,A -85,B 0,C 180,E1 27103.553,E2 27103.553} C_VEL
LIN {X 0,Y 576.024,Z 897.991,A -85,B 0,C 180,E1 27102.328,E2 27102.328} C_VEL
LIN {X 0,Y 576.096,Z 888.287,A -85,B 0,C 180,E1 27101.209,E2 27101.209} C_VEL
LIN {X 0,Y 576.195,Z 877.273,A -85,B 0,C 180,E1 27100.195,E2 27100.195} C_VEL
LIN {X 0,Y 576.276,Z 865.338,A -85,B 0,C 180,E1 27099.336,E2 27099.336} C_VEL
LIN {X 0,Y 576.421,Z 851.624,A -85,B 0,C 180,E1 27098.579,E2 27098.579} C_VEL
LIN {X 0,Y 576.524,Z 836.832,A -85,B 0,C 180,E1 27097.993,E2 27097.993} C_VEL
LIN {X 0,Y 576.587,Z 822.093,A -85,B 0,C 180,E1 27097.614,E2 27097.614} C_VEL
LIN {X 0,Y 576.647,Z 780.448,A -85,B 0,C 180,E1 27097.063,E2 27097.063} C_VEL
LIN {X 0,Y 576.539,Z 711.285,A -85,B 0,C 180,E1 27096.191,E2 27096.191} C_VEL
LIN {X 0,Y 576.366,Z 709.468,A -85,B 0,C 180,E1 27096.124,E2 27096.124} C_VEL
LIN {X 0,Y 576.583,Z 677.301,A -85,B 0,C 180,E1 27092.743,E2 27092.743} C_VEL
LIN {X 0,Y 576.867,Z 645.28,A -85,B 0,C 180,E1 27089.305,E2 27089.305} C_VEL
LIN {X 0,Y 577.18,Z 615.369,A -85,B 0,C 180,E1 27086.026,E2 27086.026} C_VEL
LIN {X 0,Y 577.51,Z 589.587,A -85,B 0,C 180,E1 27083.139,E2 27083.139} C_VEL
LIN {X 0,Y 576.16,Z 584.148,A -85,B 0,C 180,E1 27082.396,E2 27082.396} C_VEL
LIN {X 0,Y 576.146,Z 584.033,A -85,B 0,C 180,E1 27079.191,E2 27079.191} C_VEL
LIN {X 0,Y 576.137,Z 584.027,A -85,B 0,C 180,E1 27075.938,E2 27075.938} C_VEL
LIN {X 0,Y 576.147,Z 584.027,A -85,B 0,C 180,E1 27072.737,E2 27072.737} C_VEL
LIN {X 0,Y 576.138,Z 584.028,A -85,B 0,C 180,E1 27069.478,E2 27069.478} C_VEL
LIN {X 0,Y 576.155,Z 584.015,A -85,B 0,C 180,E1 27066.144,E2 27066.144} C_VEL
LIN {X 0,Y 576.156,Z 584.033,A -85,B 0,C 180,E1 27062.732,E2 27062.732} C_VEL
LIN {X 0,Y 576.134,Z 584.019,A -85,B 0,C 180,E1 27059.406,E2 27059.406} C_VEL
LIN {X 0,Y 576.151,Z 584.028,A -85,B 0,C 180,E1 27056.146,E2 27056.146} C_VEL
LIN {X 0,Y 576.129,Z 584.027,A -85,B 0,C 180,E1 27052.97,E2 27052.97} C_VEL
LIN {X 0,Y 576.15,Z 584.027,A -85,B 0,C 180,E1 27049.782,E2 27049.782} C_VEL
LIN {X 0,Y 576.128,Z 584.026,A -85,B 0,C 180,E1 27046.587,E2 27046.587} C_VEL
LIN {X 0,Y 576.156,Z 584.023,A -85,B 0,C 180,E1 27043.274,E2 27043.274} C_VEL
LIN {X 0,Y 576.15,Z 584.029,A -85,B 0,C 180,E1 27039.909,E2 27039.909} C_VEL
LIN {X 0,Y 576.137,Z 584.024,A -85,B 0,C 180,E1 27036.655,E2 27036.655} C_VEL
LIN {X 0,Y 576.158,Z 584.028,A -85,B 0,C 180,E1 27033.376,E2 27033.376} C_VEL
LIN {X 0,Y 576.122,Z 584.028,A -85,B 0,C 180,E1 27030.104,E2 27030.104} C_VEL
LIN {X 0,Y 576.156,Z 584.022,A -85,B 0,C 180,E1 27026.933,E2 27026.933} C_VEL
LIN {X 0,Y 576.118,Z 584.027,A -85,B 0,C 180,E1 27023.744,E2 27023.744} C_VEL
LIN {X 0,Y 576.157,Z 584.024,A -85,B 0,C 180,E1 27020.521,E2 27020.521} C_VEL
LIN {X 0,Y 576.117,Z 584.025,A -85,B 0,C 180,E1 27017.342,E2 27017.342} C_VEL
LIN {X 0,Y 576.158,Z 584.023,A -85,B 0,C 180,E1 27014.048,E2 27014.048} C_VEL
LIN {X 0,Y 576.133,Z 584.032,A -85,B 0,C 180,E1 27010.801,E2 27010.801} C_VEL
LIN {X 0,Y 576.129,Z 584.022,A -85,B 0,C 180,E1 27007.479,E2 27007.479} C_VEL
LIN {X 0,Y 576.157,Z 584.032,A -85,B 0,C 180,E1 27004.28,E2 27004.28} C_VEL
LIN {X 0,Y 576.113,Z 584.024,A -85,B 0,C 180,E1 27000.995,E2 27000.995} C_VEL
LIN {X 0,Y 576.161,Z 584.028,A -85,B 0,C 180,E1 26997.812,E2 26997.812} C_VEL
LIN {X 0,Y 576.108,Z 584.029,A -85,B 0,C 180,E1 26994.623,E2 26994.623} C_VEL
LIN {X 0,Y 576.16,Z 584.025,A -85,B 0,C 180,E1 26991.417,E2 26991.417} C_VEL
LIN {X 0,Y 576.105,Z 584.03,A -85,B 0,C 180,E1 26988.284,E2 26988.284} C_VEL
LIN {X 0,Y 576.161,Z 584.024,A -85,B 0,C 180,E1 26985.118,E2 26985.118} C_VEL
LIN {X 0,Y 576.103,Z 584.031,A -85,B 0,C 180,E1 26982.005,E2 26982.005} C_VEL
LIN {X 0,Y 576.161,Z 584.024,A -85,B 0,C 180,E1 26978.841,E2 26978.841} C_VEL
LIN {X 0,Y 576.102,Z 584.031,A -85,B 0,C 180,E1 26975.712,E2 26975.712} C_VEL
LIN {X 0,Y 576.16,Z 584.024,A -85,B 0,C 180,E1 26972.473,E2 26972.473} C_VEL
LIN {X 0,Y 576.11,Z 584.031,A -85,B 0,C 180,E1 26969.32,E2 26969.32} C_VEL
LIN {X 0,Y 576.139,Z 584.025,A -85,B 0,C 180,E1 26966.026,E2 26966.026} C_VEL
LIN {X 0,Y 576.115,Z 584.033,A -85,B 0,C 180,E1 26962.971,E2 26962.971} C_VEL
LIN {X 0,Y 576.122,Z 584.027,A -85,B 0,C 180,E1 26959.631,E2 26959.631} C_VEL
LIN {X 0,Y 576.138,Z 584.033,A -85,B 0,C 180,E1 26956.504,E2 26956.504} C_VEL
LIN {X 0,Y 576.104,Z 584.029,A -85,B 0,C 180,E1 26953.203,E2 26953.203} C_VEL
LIN {X 0,Y 576.16,Z 584.032,A -85,B 0,C 180,E1 26950.066,E2 26950.066} C_VEL
LIN {X 0,Y 576.098,Z 584.03,A -85,B 0,C 180,E1 26946.861,E2 26946.861} C_VEL
LIN {X 0,Y 576.158,Z 584.027,A -85,B 0,C 180,E1 26943.734,E2 26943.734} C_VEL
LIN {X 0,Y 576.195,Z 584.252,A -85,B 0,C 180,E1 26941.314,E2 26941.314} C_VEL
LIN {X 0,Y 578.897,Z 592.992,A -85,B 0,C 180,E1 26940.474,E2 26940.474} C_VEL
LIN {X 0,Y 578.298,Z 635.717,A -85,B 0,C 180,E1 26937.437,E2 26937.437} C_VEL
LIN {X 0,Y 577.843,Z 679.825,A -85,B 0,C 180,E1 26934.374,E2 26934.374} C_VEL
LIN {X 0,Y 577.804,Z 692.223,A -85,B 0,C 180,E1 26933.557,E2 26933.557} C_VEL
LIN {X 0,Y 578.372,Z 698.384,A -85,B 0,C 180,E1 26933.448,E2 26933.448} C_VEL
LIN {X 0,Y 577.841,Z 901.304,A -85,B 0,C 180,E1 26930.777,E2 26930.777} C_VEL
LIN {X 0,Y 577.676,Z 920.34,A -85,B 0,C 180,E1 26930.336,E2 26930.336} C_VEL
LIN {X 0,Y 577.502,Z 938.397,A -85,B 0,C 180,E1 26929.732,E2 26929.732} C_VEL
LIN {X 0,Y 577.246,Z 956.414,A -85,B 0,C 180,E1 26928.933,E2 26928.933} C_VEL
LIN {X 0,Y 577.027,Z 973.588,A -85,B 0,C 180,E1 26927.965,E2 26927.965} C_VEL
LIN {X 0,Y 576.798,Z 989.182,A -85,B 0,C 180,E1 26926.889,E2 26926.889} C_VEL
LIN {X 0,Y 576.571,Z 1004.113,A -85,B 0,C 180,E1 26925.644,E2 26925.644} C_VEL
LIN {X 0,Y 576.369,Z 1017.943,A -85,B 0,C 180,E1 26924.261,E2 26924.261} C_VEL
LIN {X 0,Y 576.208,Z 1030.683,A -85,B 0,C 180,E1 26922.731,E2 26922.731} C_VEL
LIN {X 0,Y 576.085,Z 1041.865,A -85,B 0,C 180,E1 26921.108,E2 26921.108} C_VEL
LIN {X 0,Y 575.999,Z 1051.509,A -85,B 0,C 180,E1 26919.391,E2 26919.391} C_VEL
LIN {X 0,Y 575.955,Z 1059.177,A -85,B 0,C 180,E1 26917.682,E2 26917.682} C_VEL
LIN {X 0,Y 575.921,Z 1065.491,A -85,B 0,C 180,E1 26915.853,E2 26915.853} C_VEL
LIN {X 0,Y 575.919,Z 1069.875,A -85,B 0,C 180,E1 26914.082,E2 26914.082} C_VEL
LIN {X 0,Y 575.917,Z 1072.789,A -85,B 0,C 180,E1 26912.189,E2 26912.189} C_VEL
LIN {X 0,Y 575.907,Z 1073.94,A -85,B 0,C 180,E1 26910.299,E2 26910.299} C_VEL
LIN {X 0,Y 575.914,Z 1073.349,A -85,B 0,C 180,E1 26908.408,E2 26908.408} C_VEL
LIN {X 0,Y 575.908,Z 1071.006,A -85,B 0,C 180,E1 26906.516,E2 26906.516} C_VEL
LIN {X 0,Y 575.919,Z 1067.098,A -85,B 0,C 180,E1 26904.721,E2 26904.721} C_VEL
LIN {X 0,Y 575.94,Z 1061.469,A -85,B 0,C 180,E1 26902.92,E2 26902.92} C_VEL
LIN {X 0,Y 575.979,Z 1054.425,A -85,B 0,C 180,E1 26901.213,E2 26901.213} C_VEL
LIN {X 0,Y 576.056,Z 1045.513,A -85,B 0,C 180,E1 26899.499,E2 26899.499} C_VEL
LIN {X 0,Y 576.157,Z 1035.149,A -85,B 0,C 180,E1 26897.879,E2 26897.879} C_VEL
LIN {X 0,Y 576.308,Z 1022.946,A -85,B 0,C 180,E1 26896.304,E2 26896.304} C_VEL
LIN {X 0,Y 576.499,Z 1009.579,A -85,B 0,C 180,E1 26894.869,E2 26894.869} C_VEL
LIN {X 0,Y 576.719,Z 994.599,A -85,B 0,C 180,E1 26893.533,E2 26893.533} C_VEL
LIN {X 0,Y 576.96,Z 978.424,A -85,B 0,C 180,E1 26892.346,E2 26892.346} C_VEL
LIN {X 0,Y 577.165,Z 962.229,A -85,B 0,C 180,E1 26891.37,E2 26891.37} C_VEL
LIN {X 0,Y 577.43,Z 944.799,A -85,B 0,C 180,E1 26890.529,E2 26890.529} C_VEL
LIN {X 0,Y 577.621,Z 926.628,A -85,B 0,C 180,E1 26889.854,E2 26889.854} C_VEL
LIN {X 0,Y 577.789,Z 908.144,A -85,B 0,C 180,E1 26889.361,E2 26889.361} C_VEL
LIN {X 0,Y 577.901,Z 888.206,A -85,B 0,C 180,E1 26889.028,E2 26889.028} C_VEL
LIN {X 0,Y 578.208,Z 694.875,A -85,B 0,C 180,E1 26886.499,E2 26886.499} C_VEL
LIN {X 0,Y 577.732,Z 690.883,A -85,B 0,C 180,E1 26886.381,E2 26886.381} C_VEL
LIN {X 0,Y 578.229,Z 642.812,A -85,B 0,C 180,E1 26883.061,E2 26883.061} C_VEL
LIN {X 0,Y 578.81,Z 599.492,A -85,B 0,C 180,E1 26879.994,E2 26879.994} C_VEL
LIN {X 0,Y 578.809,Z 592.062,A -85,B 0,C 180,E1 26879.453,E2 26879.453} C_VEL
LIN {X 0,Y 576.195,Z 584.258,A -85,B 0,C 180,E1 26878.687,E2 26878.687} C_VEL
LIN {X 0,Y 576.097,Z 584.034,A -85,B 0,C 180,E1 26875.527,E2 26875.527} C_VEL
LIN {X 0,Y 576.162,Z 584.028,A -85,B 0,C 180,E1 26872.473,E2 26872.473} C_VEL
LIN {X 0,Y 576.096,Z 584.032,A -85,B 0,C 180,E1 26869.327,E2 26869.327} C_VEL
LIN {X 0,Y 576.164,Z 584.026,A -85,B 0,C 180,E1 26866.178,E2 26866.178} C_VEL
LIN {X 0,Y 576.094,Z 584.032,A -85,B 0,C 180,E1 26863.007,E2 26863.007} C_VEL
LIN {X 0,Y 576.163,Z 584.027,A -85,B 0,C 180,E1 26859.911,E2 26859.911} C_VEL
LIN {X 0,Y 576.095,Z 584.032,A -85,B 0,C 180,E1 26856.782,E2 26856.782} C_VEL
LIN {X 0,Y 576.159,Z 584.026,A -85,B 0,C 180,E1 26853.733,E2 26853.733} C_VEL
LIN {X 0,Y 576.098,Z 584.032,A -85,B 0,C 180,E1 26850.565,E2 26850.565} C_VEL
LIN {X 0,Y 576.159,Z 584.024,A -85,B 0,C 180,E1 26847.491,E2 26847.491} C_VEL
LIN {X 0,Y 576.099,Z 584.029,A -85,B 0,C 180,E1 26844.288,E2 26844.288} C_VEL
LIN {X 0,Y 576.161,Z 584.027,A -85,B 0,C 180,E1 26841.159,E2 26841.159} C_VEL
LIN {X 0,Y 576.102,Z 584.03,A -85,B 0,C 180,E1 26837.994,E2 26837.994} C_VEL
LIN {X 0,Y 576.161,Z 584.027,A -85,B 0,C 180,E1 26834.848,E2 26834.848} C_VEL
LIN {X 0,Y 576.104,Z 584.03,A -85,B 0,C 180,E1 26831.716,E2 26831.716} C_VEL
LIN {X 0,Y 576.159,Z 584.025,A -85,B 0,C 180,E1 26828.583,E2 26828.583} C_VEL
LIN {X 0,Y 576.107,Z 584.027,A -85,B 0,C 180,E1 26825.477,E2 26825.477} C_VEL
LIN {X 0,Y 576.16,Z 584.029,A -85,B 0,C 180,E1 26822.287,E2 26822.287} C_VEL
LIN {X 0,Y 576.111,Z 584.027,A -85,B 0,C 180,E1 26819.105,E2 26819.105} C_VEL
LIN {X 0,Y 576.156,Z 584.03,A -85,B 0,C 180,E1 26815.82,E2 26815.82} C_VEL
LIN {X 0,Y 576.122,Z 584.027,A -85,B 0,C 180,E1 26812.621,E2 26812.621} C_VEL
LIN {X 0,Y 576.129,Z 584.031,A -85,B 0,C 180,E1 26809.197,E2 26809.197} C_VEL
LIN {X 0,Y 576.158,Z 584.022,A -85,B 0,C 180,E1 26805.95,E2 26805.95} C_VEL
LIN {X 0,Y 576.158,Z 584.031,A -85,B 0,C 180,E1 26803.339,E2 26803.339} C_VEL
LIN {X 0,Y 575.155,Z 584.151,A -85,B 0,C 180,E1 26802.573,E2 26802.573} C_VEL
LIN {X 0,Y 568.702,Z 584.953,A -85,B 0,C 180,E1 26800.424,E2 26800.424} C_VEL
LIN {X 0,Y 568.207,Z 585.014,A -85,B 0,C 180,E1 26799.864,E2 26799.864} C_VEL
LIN {X 0,Y 568.188,Z 585.016,A -85,B 0,C 180,E1 26796.565,E2 26796.565} C_VEL
LIN {X 0,Y 568.22,Z 585.016,A -85,B 0,C 180,E1 26793.339,E2 26793.339} C_VEL
LIN {X 0,Y 568.184,Z 585.018,A -85,B 0,C 180,E1 26790.131,E2 26790.131} C_VEL
LIN {X 0,Y 568.217,Z 585.02,A -85,B 0,C 180,E1 26786.887,E2 26786.887} C_VEL
LIN {X 0,Y 568.186,Z 585.018,A -85,B 0,C 180,E1 26783.627,E2 26783.627} C_VEL
LIN {X 0,Y 568.223,Z 585.02,A -85,B 0,C 180,E1 26780.301,E2 26780.301} C_VEL
LIN {X 0,Y 568.22,Z 585.185,A -85,B 0,C 180,E1 26777.832,E2 26777.832} C_VEL
LIN {X 0,Y 569.938,Z 592.58,A -85,B 0,C 180,E1 26776.828,E2 26776.828} C_VEL
LIN {X 0,Y 569.457,Z 621.667,A -85,B 0,C 180,E1 26773.518,E2 26773.518} C_VEL
LIN {X 0,Y 569.054,Z 652.075,A -85,B 0,C 180,E1 26770.153,E2 26770.153} C_VEL
LIN {X 0,Y 568.715,Z 683.053,A -85,B 0,C 180,E1 26766.791,E2 26766.791} C_VEL
LIN {X 0,Y 568.518,Z 710.002,A -85,B 0,C 180,E1 26763.948,E2 26763.948} C_VEL
LIN {X 0,Y 568.987,Z 716.711,A -85,B 0,C 180,E1 26763.834,E2 26763.834} C_VEL
LIN {X 0,Y 568.767,Z 821.372,A -85,B 0,C 180,E1 26762.483,E2 26762.483} C_VEL
LIN {X 0,Y 568.69,Z 836.358,A -85,B 0,C 180,E1 26762.101,E2 26762.101} C_VEL
LIN {X 0,Y 568.563,Z 850.422,A -85,B 0,C 180,E1 26761.545,E2 26761.545} C_VEL
LIN {X 0,Y 568.425,Z 863.129,A -85,B 0,C 180,E1 26760.863,E2 26760.863} C_VEL
LIN {X 0,Y 568.278,Z 875.728,A -85,B 0,C 180,E1 26759.979,E2 26759.979} C_VEL
LIN {X 0,Y 568.163,Z 887.171,A -85,B 0,C 180,E1 26758.944,E2 26758.944} C_VEL
LIN {X 0,Y 568.064,Z 897.135,A -85,B 0,C 180,E1 26757.803,E2 26757.803} C_VEL
LIN {X 0,Y 567.988,Z 905.652,A -85,B 0,C 180,E1 26756.56,E2 26756.56} C_VEL
LIN {X 0,Y 567.947,Z 912.769,A -85,B 0,C 180,E1 26755.191,E2 26755.191} C_VEL
LIN {X 0,Y 567.925,Z 918.141,A -85,B 0,C 180,E1 26753.776,E2 26753.776} C_VEL
LIN {X 0,Y 567.919,Z 921.935,A -85,B 0,C 180,E1 26752.242,E2 26752.242} C_VEL
LIN {X 0,Y 567.916,Z 923.745,A -85,B 0,C 180,E1 26750.724,E2 26750.724} C_VEL
LIN {X 0,Y 567.916,Z 923.769,A -85,B 0,C 180,E1 26749.222,E2 26749.222} C_VEL
LIN {X 0,Y 567.917,Z 922.05,A -85,B 0,C 180,E1 26747.733,E2 26747.733} C_VEL
LIN {X 0,Y 567.922,Z 918.507,A -85,B 0,C 180,E1 26746.256,E2 26746.256} C_VEL
LIN {X 0,Y 567.944,Z 913.45,A -85,B 0,C 180,E1 26744.869,E2 26744.869} C_VEL
LIN {X 0,Y 567.986,Z 906.161,A -85,B 0,C 180,E1 26743.436,E2 26743.436} C_VEL
LIN {X 0,Y 568.057,Z 897.791,A -85,B 0,C 180,E1 26742.194,E2 26742.194} C_VEL
LIN {X 0,Y 568.15,Z 888.05,A -85,B 0,C 180,E1 26741.059,E2 26741.059} C_VEL
LIN {X 0,Y 568.28,Z 876.345,A -85,B 0,C 180,E1 26739.98,E2 26739.98} C_VEL
LIN {X 0,Y 568.414,Z 863.297,A -85,B 0,C 180,E1 26739.058,E2 26739.058} C_VEL
LIN {X 0,Y 568.566,Z 849.93,A -85,B 0,C 180,E1 26738.342,E2 26738.342} C_VEL
LIN {X 0,Y 568.699,Z 835.435,A -85,B 0,C 180,E1 26737.78,E2 26737.78} C_VEL
LIN {X 0,Y 568.78,Z 819.74,A -85,B 0,C 180,E1 26737.395,E2 26737.395} C_VEL
LIN {X 0,Y 568.778,Z 712.196,A -85,B 0,C 180,E1 26736.013,E2 26736.013} C_VEL
LIN {X 0,Y 568.491,Z 709.491,A -85,B 0,C 180,E1 26735.931,E2 26735.931} C_VEL
LIN {X 0,Y 568.766,Z 677.484,A -85,B 0,C 180,E1 26732.519,E2 26732.519} C_VEL
LIN {X 0,Y 569.12,Z 646.035,A -85,B 0,C 180,E1 26729.094,E2 26729.094} C_VEL
LIN {X 0,Y 569.51,Z 617.036,A -85,B 0,C 180,E1 26725.872,E2 26725.872} C_VEL
LIN {X 0,Y 569.901,Z 591.799,A -85,B 0,C 180,E1 26722.996,E2 26722.996} C_VEL
LIN {X 0,Y 568.221,Z 585.173,A -85,B 0,C 180,E1 26722.086,E2 26722.086} C_VEL
LIN {X 0,Y 568.209,Z 585.018,A -85,B 0,C 180,E1 26718.839,E2 26718.839} C_VEL
LIN {X 0,Y 568.21,Z 585.02,A -85,B 0,C 180,E1 26715.53,E2 26715.53} C_VEL
LIN {X 0,Y 568.206,Z 585.013,A -85,B 0,C 180,E1 26712.064,E2 26712.064} C_VEL
LIN {X 0,Y 568.211,Z 585.018,A -85,B 0,C 180,E1 26708.746,E2 26708.746} C_VEL
LIN {X 0,Y 568.192,Z 585.007,A -85,B 0,C 180,E1 26705.462,E2 26705.462} C_VEL
LIN {X 0,Y 568.211,Z 585.014,A -85,B 0,C 180,E1 26702.205,E2 26702.205} C_VEL
LIN {X 0,Y 568.198,Z 585.011,A -85,B 0,C 180,E1 26698.962,E2 26698.962} C_VEL
LIN {X 0,Y 568.215,Z 585.012,A -85,B 0,C 180,E1 26695.608,E2 26695.608} C_VEL
LIN {X 0,Y 568.22,Z 585.019,A -85,B 0,C 180,E1 26692.24,E2 26692.24} C_VEL
LIN {X 0,Y 568.193,Z 585.015,A -85,B 0,C 180,E1 26688.976,E2 26688.976} C_VEL
LIN {X 0,Y 568.212,Z 585.016,A -85,B 0,C 180,E1 26685.686,E2 26685.686} C_VEL
LIN {X 0,Y 568.189,Z 585.017,A -85,B 0,C 180,E1 26682.495,E2 26682.495} C_VEL
LIN {X 0,Y 568.216,Z 585.013,A -85,B 0,C 180,E1 26679.263,E2 26679.263} C_VEL
LIN {X 0,Y 568.191,Z 585.02,A -85,B 0,C 180,E1 26675.998,E2 26675.998} C_VEL
LIN {X 0,Y 568.203,Z 585.01,A -85,B 0,C 180,E1 26672.579,E2 26672.579} C_VEL
LIN {X 0,Y 568.222,Z 585.019,A -85,B 0,C 180,E1 26669.287,E2 26669.287} C_VEL
LIN {X 0,Y 568.182,Z 585.011,A -85,B 0,C 180,E1 26665.941,E2 26665.941} C_VEL
LIN {X 0,Y 568.218,Z 585.016,A -85,B 0,C 180,E1 26662.771,E2 26662.771} C_VEL
LIN {X 0,Y 568.179,Z 585.017,A -85,B 0,C 180,E1 26659.534,E2 26659.534} C_VEL
LIN {X 0,Y 568.221,Z 585.01,A -85,B 0,C 180,E1 26656.247,E2 26656.247} C_VEL
LIN {X 0,Y 568.183,Z 585.021,A -85,B 0,C 180,E1 26653.018,E2 26653.018} C_VEL
LIN {X 0,Y 568.195,Z 585.008,A -85,B 0,C 180,E1 26649.624,E2 26649.624} C_VEL
LIN {X 0,Y 568.221,Z 585.02,A -85,B 0,C 180,E1 26646.365,E2 26646.365} C_VEL
LIN {X 0,Y 568.178,Z 585.015,A -85,B 0,C 180,E1 26643.127,E2 26643.127} C_VEL
LIN {X 0,Y 568.223,Z 585.014,A -85,B 0,C 180,E1 26639.899,E2 26639.899} C_VEL
LIN {X 0,Y 568.17,Z 585.018,A -85,B 0,C 180,E1 26636.671,E2 26636.671} C_VEL
LIN {X 0,Y 568.221,Z 585.008,A -85,B 0,C 180,E1 26633.433,E2 26633.433} C_VEL
LIN {X 0,Y 568.167,Z 585.019,A -85,B 0,C 180,E1 26630.274,E2 26630.274} C_VEL
LIN {X 0,Y 568.215,Z 585.011,A -85,B 0,C 180,E1 26626.983,E2 26626.983} C_VEL
LIN {X 0,Y 568.173,Z 585.019,A -85,B 0,C 180,E1 26623.857,E2 26623.857} C_VEL
LIN {X 0,Y 568.189,Z 585.013,A -85,B 0,C 180,E1 26620.467,E2 26620.467} C_VEL
LIN {X 0,Y 568.215,Z 585.021,A -85,B 0,C 180,E1 26617.225,E2 26617.225} C_VEL
LIN {X 0,Y 568.17,Z 585.014,A -85,B 0,C 180,E1 26614.012,E2 26614.012} C_VEL
LIN {X 0,Y 568.224,Z 585.019,A -85,B 0,C 180,E1 26610.829,E2 26610.829} C_VEL
LIN {X 0,Y 568.164,Z 585.018,A -85,B 0,C 180,E1 26607.641,E2 26607.641} C_VEL
LIN {X 0,Y 568.224,Z 585.019,A -85,B 0,C 180,E1 26604.502,E2 26604.502} C_VEL
LIN {X 0,Y 568.156,Z 585.018,A -85,B 0,C 180,E1 26601.337,E2 26601.337} C_VEL
LIN {X 0,Y 568.224,Z 585.018,A -85,B 0,C 180,E1 26598.172,E2 26598.172} C_VEL
LIN {X 0,Y 568.157,Z 585.019,A -85,B 0,C 180,E1 26595.028,E2 26595.028} C_VEL
LIN {X 0,Y 568.224,Z 585.016,A -85,B 0,C 180,E1 26591.828,E2 26591.828} C_VEL
LIN {X 0,Y 568.158,Z 585.021,A -85,B 0,C 180,E1 26588.663,E2 26588.663} C_VEL
LIN {X 0,Y 568.224,Z 585.016,A -85,B 0,C 180,E1 26585.442,E2 26585.442} C_VEL
LIN {X 0,Y 568.168,Z 585.02,A -85,B 0,C 180,E1 26582.224,E2 26582.224} C_VEL
LIN {X 0,Y 568.263,Z 585.337,A -85,B 0,C 180,E1 26581.71,E2 26581.71} C_VEL
LIN {X 0,Y 571.665,Z 595.547,A -85,B 0,C 180,E1 26580.712,E2 26580.712} C_VEL
LIN {X 0,Y 570.925,Z 638.08,A -85,B 0,C 180,E1 26577.652,E2 26577.652} C_VEL
LIN {X 0,Y 570.338,Z 682.188,A -85,B 0,C 180,E1 26574.55,E2 26574.55} C_VEL
LIN {X 0,Y 570.306,Z 692.219,A -85,B 0,C 180,E1 26573.886,E2 26573.886} C_VEL
LIN {X 0,Y 571.03,Z 699.148,A -85,B 0,C 180,E1 26573.758,E2 26573.758} C_VEL
LIN {X 0,Y 570.358,Z 901.304,A -85,B 0,C 180,E1 26571.062,E2 26571.062} C_VEL
LIN {X 0,Y 570.156,Z 920.339,A -85,B 0,C 180,E1 26570.616,E2 26570.616} C_VEL
LIN {X 0,Y 569.932,Z 938.395,A -85,B 0,C 180,E1 26570.005,E2 26570.005} C_VEL
LIN {X 0,Y 569.622,Z 956.257,A -85,B 0,C 180,E1 26569.204,E2 26569.204} C_VEL
LIN {X 0,Y 569.348,Z 972.774,A -85,B 0,C 180,E1 26568.269,E2 26568.269} C_VEL
LIN {X 0,Y 569.054,Z 988.629,A -85,B 0,C 180,E1 26567.169,E2 26567.169} C_VEL
LIN {X 0,Y 568.768,Z 1003.557,A -85,B 0,C 180,E1 26565.917,E2 26565.917} C_VEL
LIN {X 0,Y 568.523,Z 1017.017,A -85,B 0,C 180,E1 26564.566,E2 26564.566} C_VEL
LIN {X 0,Y 568.307,Z 1029.909,A -85,B 0,C 180,E1 26563.015,E2 26563.015} C_VEL
LIN {X 0,Y 568.141,Z 1041.227,A -85,B 0,C 180,E1 26561.368,E2 26561.368} C_VEL
LIN {X 0,Y 568.032,Z 1050.992,A -85,B 0,C 180,E1 26559.627,E2 26559.627} C_VEL
LIN {X 0,Y 567.963,Z 1058.772,A -85,B 0,C 180,E1 26557.893,E2 26557.893} C_VEL
LIN {X 0,Y 567.932,Z 1065.109,A -85,B 0,C 180,E1 26556.064,E2 26556.064} C_VEL
LIN {X 0,Y 567.92,Z 1069.875,A -85,B 0,C 180,E1 26554.14,E2 26554.14} C_VEL
LIN {X 0,Y 567.916,Z 1072.79,A -85,B 0,C 180,E1 26552.22,E2 26552.22} C_VEL
LIN {X 0,Y 567.907,Z 1073.94,A -85,B 0,C 180,E1 26550.303,E2 26550.303} C_VEL
LIN {X 0,Y 567.914,Z 1073.349,A -85,B 0,C 180,E1 26548.386,E2 26548.386} C_VEL
LIN {X 0,Y 567.909,Z 1071.005,A -85,B 0,C 180,E1 26546.467,E2 26546.467} C_VEL
LIN {X 0,Y 567.923,Z 1067.098,A -85,B 0,C 180,E1 26544.646,E2 26544.646} C_VEL
LIN {X 0,Y 567.947,Z 1061.469,A -85,B 0,C 180,E1 26542.82,E2 26542.82} C_VEL
LIN {X 0,Y 568.001,Z 1054.425,A -85,B 0,C 180,E1 26541.089,E2 26541.089} C_VEL
LIN {X 0,Y 568.099,Z 1045.514,A -85,B 0,C 180,E1 26539.351,E2 26539.351} C_VEL
LIN {X 0,Y 568.23,Z 1035.15,A -85,B 0,C 180,E1 26537.707,E2 26537.707} C_VEL
LIN {X 0,Y 568.413,Z 1023.349,A -85,B 0,C 180,E1 26536.159,E2 26536.159} C_VEL
LIN {X 0,Y 568.65,Z 1010.085,A -85,B 0,C 180,E1 26534.708,E2 26534.708} C_VEL
LIN {X 0,Y 568.929,Z 995.228,A -85,B 0,C 180,E1 26533.354,E2 26533.354} C_VEL
LIN {X 0,Y 569.235,Z 979.23,A -85,B 0,C 180,E1 26532.151,E2 26532.151} C_VEL
LIN {X 0,Y 569.512,Z 962.142,A -85,B 0,C 180,E1 26531.106,E2 26531.106} C_VEL
LIN {X 0,Y 569.837,Z 944.801,A -85,B 0,C 180,E1 26530.259,E2 26530.259} C_VEL
LIN {X 0,Y 570.081,Z 926.631,A -85,B 0,C 180,E1 26529.576,E2 26529.576} C_VEL
LIN {X 0,Y 570.294,Z 908.143,A -85,B 0,C 180,E1 26529.077,E2 26529.077} C_VEL
LIN {X 0,Y 570.432,Z 888,A -85,B 0,C 180,E1 26528.738,E2 26528.738} C_VEL
LIN {X 0,Y 570.876,Z 696.003,A -85,B 0,C 180,E1 26526.193,E2 26526.193} C_VEL
LIN {X 0,Y 570.239,Z 691.329,A -85,B 0,C 180,E1 26526.079,E2 26526.079} C_VEL
LIN {X 0,Y 570.853,Z 643.6,A -85,B 0,C 180,E1 26522.74,E2 26522.74} C_VEL
LIN {X 0,Y 571.586,Z 600.279,A -85,B 0,C 180,E1 26519.633,E2 26519.633} C_VEL
LIN {X 0,Y 571.466,Z 594.688,A -85,B 0,C 180,E1 26519.213,E2 26519.213} C_VEL
LIN {X 0,Y 568.261,Z 585.323,A -85,B 0,C 180,E1 26518.288,E2 26518.288} C_VEL
LIN {X 0,Y 568.202,Z 585.014,A -85,B 0,C 180,E1 26516.821,E2 26516.821} C_VEL
LIN {X 0,Y 568.167,Z 585.024,A -85,B 0,C 180,E1 26513.626,E2 26513.626} C_VEL
LIN {X 0,Y 568.225,Z 585.015,A -85,B 0,C 180,E1 26510.433,E2 26510.433} C_VEL
LIN {X 0,Y 568.157,Z 585.021,A -85,B 0,C 180,E1 26507.21,E2 26507.21} C_VEL
LIN {X 0,Y 568.223,Z 585.016,A -85,B 0,C 180,E1 26504.116,E2 26504.116} C_VEL
LIN {X 0,Y 568.155,Z 585.021,A -85,B 0,C 180,E1 26500.894,E2 26500.894} C_VEL
LIN {X 0,Y 568.225,Z 585.015,A -85,B 0,C 180,E1 26497.759,E2 26497.759} C_VEL
LIN {X 0,Y 568.157,Z 585.02,A -85,B 0,C 180,E1 26494.64,E2 26494.64} C_VEL
LIN {X 0,Y 568.225,Z 585.016,A -85,B 0,C 180,E1 26491.507,E2 26491.507} C_VEL
LIN {X 0,Y 568.159,Z 585.018,A -85,B 0,C 180,E1 26488.368,E2 26488.368} C_VEL
LIN {X 0,Y 568.223,Z 585.018,A -85,B 0,C 180,E1 26485.203,E2 26485.203} C_VEL
LIN {X 0,Y 568.163,Z 585.018,A -85,B 0,C 180,E1 26482.014,E2 26482.014} C_VEL
LIN {X 0,Y 568.222,Z 585.017,A -85,B 0,C 180,E1 26478.784,E2 26478.784} C_VEL
LIN {X 0,Y 568.171,Z 585.016,A -85,B 0,C 180,E1 26475.619,E2 26475.619} C_VEL
LIN {X 0,Y 568.195,Z 585.022,A -85,B 0,C 180,E1 26472.294,E2 26472.294} C_VEL
LIN {X 0,Y 568.191,Z 585.011,A -85,B 0,C 180,E1 26469.112,E2 26469.112} C_VEL
LIN {X 0,Y 568.174,Z 585.018,A -85,B 0,C 180,E1 26465.757,E2 26465.757} C_VEL
LIN {X 0,Y 568.221,Z 585.014,A -85,B 0,C 180,E1 26462.521,E2 26462.521} C_VEL
LIN {X 0,Y 568.172,Z 585.017,A -85,B 0,C 180,E1 26459.294,E2 26459.294} C_VEL
LIN {X 0,Y 568.22,Z 585.018,A -85,B 0,C 180,E1 26456.065,E2 26456.065} C_VEL
LIN {X 0,Y 568.175,Z 585.017,A -85,B 0,C 180,E1 26452.822,E2 26452.822} C_VEL
LIN {X 0,Y 568.219,Z 585.02,A -85,B 0,C 180,E1 26449.558,E2 26449.558} C_VEL
LIN {X 0,Y 568.193,Z 585.012,A -85,B 0,C 180,E1 26446.256,E2 26446.256} C_VEL
LIN {X 0,Y 568.187,Z 585.017,A -85,B 0,C 180,E1 26442.851,E2 26442.851} C_VEL
LIN {X 0,Y 568.207,Z 585.014,A -85,B 0,C 180,E1 26439.864,E2 26439.864} C_VEL
LIN {X 0,Y 567.263,Z 585.138,A -85,B 0,C 180,E1 26439.087,E2 26439.087} C_VEL
LIN {X 0,Y 560.689,Z 585.954,A -85,B 0,C 180,E1 26436.85,E2 26436.85} C_VEL
LIN {X 0,Y 560.241,Z 586.004,A -85,B 0,C 180,E1 26436.338,E2 26436.338} C_VEL
LIN {X 0,Y 560.28,Z 586.008,A -85,B 0,C 180,E1 26433.045,E2 26433.045} C_VEL
LIN {X 0,Y 560.249,Z 586.005,A -85,B 0,C 180,E1 26429.744,E2 26429.744} C_VEL
LIN {X 0,Y 560.273,Z 586.008,A -85,B 0,C 180,E1 26426.411,E2 26426.411} C_VEL
LIN {X 0,Y 560.28,Z 586.006,A -85,B 0,C 180,E1 26423.029,E2 26423.029} C_VEL
LIN {X 0,Y 560.252,Z 586.012,A -85,B 0,C 180,E1 26419.755,E2 26419.755} C_VEL
LIN {X 0,Y 560.315,Z 586.26,A -85,B 0,C 180,E1 26418.155,E2 26418.155} C_VEL
LIN {X 0,Y 562.418,Z 595.253,A -85,B 0,C 180,E1 26416.943,E2 26416.943} C_VEL
LIN {X 0,Y 561.761,Z 624.125,A -85,B 0,C 180,E1 26413.58,E2 26413.58} C_VEL
LIN {X 0,Y 561.276,Z 654.049,A -85,B 0,C 180,E1 26410.225,E2 26410.225} C_VEL
LIN {X 0,Y 560.884,Z 684.052,A -85,B 0,C 180,E1 26406.924,E2 26406.924} C_VEL
LIN {X 0,Y 560.63,Z 709.869,A -85,B 0,C 180,E1 26404.154,E2 26404.154} C_VEL
LIN {X 0,Y 561.219,Z 717.036,A -85,B 0,C 180,E1 26404.026,E2 26404.026} C_VEL
LIN {X 0,Y 560.954,Z 821.389,A -85,B 0,C 180,E1 26402.66,E2 26402.66} C_VEL
LIN {X 0,Y 560.863,Z 836.013,A -85,B 0,C 180,E1 26402.284,E2 26402.284} C_VEL
LIN {X 0,Y 560.702,Z 850.774,A -85,B 0,C 180,E1 26401.694,E2 26401.694} C_VEL
LIN {X 0,Y 560.53,Z 863.852,A -85,B 0,C 180,E1 26400.972,E2 26400.972} C_VEL
LIN {X 0,Y 560.355,Z 876.367,A -85,B 0,C 180,E1 26400.071,E2 26400.071} C_VEL
LIN {X 0,Y 560.211,Z 887.783,A -85,B 0,C 180,E1 26399.008,E2 26399.008} C_VEL
LIN {X 0,Y 560.096,Z 897.356,A -85,B 0,C 180,E1 26397.886,E2 26397.886} C_VEL
LIN {X 0,Y 560.002,Z 906.239,A -85,B 0,C 180,E1 26396.553,E2 26396.553} C_VEL
LIN {X 0,Y 559.951,Z 913.357,A -85,B 0,C 180,E1 26395.134,E2 26395.134} C_VEL
LIN {X 0,Y 559.926,Z 918.558,A -85,B 0,C 180,E1 26393.69,E2 26393.69} C_VEL
LIN {X 0,Y 559.919,Z 921.989,A -85,B 0,C 180,E1 26392.245,E2 26392.245} C_VEL
LIN {X 0,Y 559.916,Z 923.799,A -85,B 0,C 180,E1 26390.654,E2 26390.654} C_VEL
LIN {X 0,Y 559.916,Z 923.731,A -85,B 0,C 180,E1 26389.151,E2 26389.151} C_VEL
LIN {X 0,Y 559.917,Z 922.002,A -85,B 0,C 180,E1 26387.672,E2 26387.672} C_VEL
LIN {X 0,Y 559.927,Z 918.244,A -85,B 0,C 180,E1 26386.114,E2 26386.114} C_VEL
LIN {X 0,Y 559.952,Z 912.965,A -85,B 0,C 180,E1 26384.688,E2 26384.688} C_VEL
LIN {X 0,Y 560.002,Z 906.008,A -85,B 0,C 180,E1 26383.316,E2 26383.316} C_VEL
LIN {X 0,Y 560.101,Z 896.805,A -85,B 0,C 180,E1 26381.951,E2 26381.951} C_VEL
LIN {X 0,Y 560.228,Z 886.823,A -85,B 0,C 180,E1 26380.801,E2 26380.801} C_VEL
LIN {X 0,Y 560.373,Z 874.702,A -85,B 0,C 180,E1 26379.707,E2 26379.707} C_VEL
LIN {X 0,Y 560.554,Z 861.979,A -85,B 0,C 180,E1 26378.82,E2 26378.82} C_VEL
LIN {X 0,Y 560.733,Z 848.21,A -85,B 0,C 180,E1 26378.098,E2 26378.098} C_VEL
LIN {X 0,Y 560.876,Z 834.1,A -85,B 0,C 180,E1 26377.567,E2 26377.567} C_VEL
LIN {X 0,Y 560.975,Z 818.975,A -85,B 0,C 180,E1 26377.204,E2 26377.204} C_VEL
LIN {X 0,Y 560.996,Z 712.846,A -85,B 0,C 180,E1 26375.824,E2 26375.824} C_VEL
LIN {X 0,Y 560.617,Z 709.517,A -85,B 0,C 180,E1 26375.732,E2 26375.732} C_VEL
LIN {X 0,Y 560.949,Z 678.227,A -85,B 0,C 180,E1 26372.349,E2 26372.349} C_VEL
LIN {X 0,Y 561.371,Z 647.704,A -85,B 0,C 180,E1 26368.979,E2 26368.979} C_VEL
LIN {X 0,Y 561.844,Z 618.703,A -85,B 0,C 180,E1 26365.713,E2 26365.713} C_VEL
LIN {X 0,Y 562.31,Z 594.036,A -85,B 0,C 180,E1 26362.84,E2 26362.84} C_VEL
LIN {X 0,Y 560.292,Z 586.131,A -85,B 0,C 180,E1 26361.74,E2 26361.74} C_VEL
LIN {X 0,Y 560.272,Z 586.005,A -85,B 0,C 180,E1 26358.366,E2 26358.366} C_VEL
LIN {X 0,Y 560.267,Z 586.008,A -85,B 0,C 180,E1 26355.003,E2 26355.003} C_VEL
LIN {X 0,Y 560.259,Z 586.005,A -85,B 0,C 180,E1 26351.701,E2 26351.701} C_VEL
LIN {X 0,Y 560.273,Z 586.003,A -85,B 0,C 180,E1 26348.4,E2 26348.4} C_VEL
LIN {X 0,Y 560.269,Z 585.999,A -85,B 0,C 180,E1 26345.038,E2 26345.038} C_VEL
LIN {X 0,Y 560.265,Z 586.002,A -85,B 0,C 180,E1 26341.621,E2 26341.621} C_VEL
LIN {X 0,Y 560.273,Z 586.001,A -85,B 0,C 180,E1 26338.349,E2 26338.349} C_VEL
LIN {X 0,Y 560.254,Z 586.005,A -85,B 0,C 180,E1 26335.049,E2 26335.049} C_VEL
LIN {X 0,Y 560.276,Z 586.002,A -85,B 0,C 180,E1 26331.738,E2 26331.738} C_VEL
LIN {X 0,Y 560.263,Z 586.01,A -85,B 0,C 180,E1 26328.397,E2 26328.397} C_VEL
LIN {X 0,Y 560.261,Z 586.002,A -85,B 0,C 180,E1 26324.969,E2 26324.969} C_VEL
LIN {X 0,Y 560.278,Z 586.002,A -85,B 0,C 180,E1 26321.732,E2 26321.732} C_VEL
LIN {X 0,Y 560.248,Z 586.005,A -85,B 0,C 180,E1 26318.42,E2 26318.42} C_VEL
LIN {X 0,Y 560.276,Z 586,A -85,B 0,C 180,E1 26315.18,E2 26315.18} C_VEL
LIN {X 0,Y 560.245,Z 586.004,A -85,B 0,C 180,E1 26312.009,E2 26312.009} C_VEL
LIN {X 0,Y 560.28,Z 586,A -85,B 0,C 180,E1 26308.689,E2 26308.689} C_VEL
LIN {X 0,Y 560.263,Z 586.003,A -85,B 0,C 180,E1 26305.361,E2 26305.361} C_VEL
LIN {X 0,Y 560.251,Z 586.004,A -85,B 0,C 180,E1 26302.011,E2 26302.011} C_VEL
LIN {X 0,Y 560.281,Z 586,A -85,B 0,C 180,E1 26298.737,E2 26298.737} C_VEL
LIN {X 0,Y 560.239,Z 586.004,A -85,B 0,C 180,E1 26295.422,E2 26295.422} C_VEL
LIN {X 0,Y 560.28,Z 586.002,A -85,B 0,C 180,E1 26292.157,E2 26292.157} C_VEL
LIN {X 0,Y 560.24,Z 586.003,A -85,B 0,C 180,E1 26288.933,E2 26288.933} C_VEL
LIN {X 0,Y 560.271,Z 586.001,A -85,B 0,C 180,E1 26285.633,E2 26285.633} C_VEL
LIN {X 0,Y 560.264,Z 586.01,A -85,B 0,C 180,E1 26282.353,E2 26282.353} C_VEL
LIN {X 0,Y 560.243,Z 586.001,A -85,B 0,C 180,E1 26279.08,E2 26279.08} C_VEL
LIN {X 0,Y 560.284,Z 586.006,A -85,B 0,C 180,E1 26275.804,E2 26275.804} C_VEL
LIN {X 0,Y 560.231,Z 586,A -85,B 0,C 180,E1 26272.617,E2 26272.617} C_VEL
LIN {X 0,Y 560.284,Z 586.005,A -85,B 0,C 180,E1 26269.408,E2 26269.408} C_VEL
LIN {X 0,Y 560.227,Z 586.005,A -85,B 0,C 180,E1 26266.269,E2 26266.269} C_VEL
LIN {X 0,Y 560.284,Z 586.004,A -85,B 0,C 180,E1 26263.044,E2 26263.044} C_VEL
LIN {X 0,Y 560.227,Z 586.007,A -85,B 0,C 180,E1 26259.848,E2 26259.848} C_VEL
LIN {X 0,Y 560.274,Z 586.003,A -85,B 0,C 180,E1 26256.549,E2 26256.549} C_VEL
LIN {X 0,Y 560.237,Z 586.007,A -85,B 0,C 180,E1 26253.387,E2 26253.387} C_VEL
LIN {X 0,Y 560.243,Z 586.004,A -85,B 0,C 180,E1 26250.019,E2 26250.019} C_VEL
LIN {X 0,Y 560.273,Z 586.011,A -85,B 0,C 180,E1 26246.823,E2 26246.823} C_VEL
LIN {X 0,Y 560.225,Z 586.008,A -85,B 0,C 180,E1 26243.536,E2 26243.536} C_VEL
LIN {X 0,Y 560.288,Z 586.01,A -85,B 0,C 180,E1 26240.425,E2 26240.425} C_VEL
LIN {X 0,Y 560.219,Z 586.009,A -85,B 0,C 180,E1 26237.184,E2 26237.184} C_VEL
LIN {X 0,Y 560.287,Z 586.006,A -85,B 0,C 180,E1 26234.014,E2 26234.014} C_VEL
LIN {X 0,Y 560.218,Z 586.01,A -85,B 0,C 180,E1 26230.786,E2 26230.786} C_VEL
LIN {X 0,Y 560.285,Z 586.005,A -85,B 0,C 180,E1 26227.595,E2 26227.595} C_VEL
LIN {X 0,Y 560.222,Z 586.013,A -85,B 0,C 180,E1 26224.456,E2 26224.456} C_VEL
LIN {X 0,Y 560.261,Z 586.19,A -85,B 0,C 180,E1 26222.129,E2 26222.129} C_VEL
LIN {X 0,Y 562.105,Z 591.531,A -85,B 0,C 180,E1 26221.567,E2 26221.567} C_VEL
LIN {X 0,Y 564.432,Z 598.698,A -85,B 0,C 180,E1 26220.912,E2 26220.912} C_VEL
LIN {X 0,Y 563.546,Z 641.231,A -85,B 0,C 180,E1 26217.816,E2 26217.816} C_VEL
LIN {X 0,Y 562.826,Z 685.339,A -85,B 0,C 180,E1 26214.676,E2 26214.676} C_VEL
LIN {X 0,Y 562.835,Z 692.286,A -85,B 0,C 180,E1 26214.222,E2 26214.222} C_VEL
LIN {X 0,Y 563.705,Z 700.108,A -85,B 0,C 180,E1 26214.073,E2 26214.073} C_VEL
LIN {X 0,Y 562.89,Z 901.304,A -85,B 0,C 180,E1 26211.355,E2 26211.355} C_VEL
LIN {X 0,Y 562.651,Z 920.319,A -85,B 0,C 180,E1 26210.905,E2 26210.905} C_VEL
LIN {X 0,Y 562.376,Z 938.394,A -85,B 0,C 180,E1 26210.286,E2 26210.286} C_VEL
LIN {X 0,Y 562.011,Z 956.142,A -85,B 0,C 180,E1 26209.481,E2 26209.481} C_VEL
LIN {X 0,Y 561.665,Z 972.772,A -85,B 0,C 180,E1 26208.528,E2 26208.528} C_VEL
LIN {X 0,Y 561.31,Z 988.627,A -85,B 0,C 180,E1 26207.413,E2 26207.413} C_VEL
LIN {X 0,Y 560.953,Z 1003.912,A -85,B 0,C 180,E1 26206.111,E2 26206.111} C_VEL
LIN {X 0,Y 560.643,Z 1017.942,A -85,B 0,C 180,E1 26204.67,E2 26204.67} C_VEL
LIN {X 0,Y 560.379,Z 1031.086,A -85,B 0,C 180,E1 26203.043,E2 26203.043} C_VEL
LIN {X 0,Y 560.187,Z 1041.865,A -85,B 0,C 180,E1 26201.427,E2 26201.427} C_VEL
LIN {X 0,Y 560.056,Z 1051.508,A -85,B 0,C 180,E1 26199.661,E2 26199.661} C_VEL
LIN {X 0,Y 559.974,Z 1059.177,A -85,B 0,C 180,E1 26197.903,E2 26197.903} C_VEL
LIN {X 0,Y 559.935,Z 1065.411,A -85,B 0,C 180,E1 26196.048,E2 26196.048} C_VEL
LIN {X 0,Y 559.921,Z 1069.876,A -85,B 0,C 180,E1 26194.199,E2 26194.199} C_VEL
LIN {X 0,Y 559.915,Z 1072.791,A -85,B 0,C 180,E1 26192.252,E2 26192.252} C_VEL
LIN {X 0,Y 559.908,Z 1073.94,A -85,B 0,C 180,E1 26190.307,E2 26190.307} C_VEL
LIN {X 0,Y 559.913,Z 1073.348,A -85,B 0,C 180,E1 26188.363,E2 26188.363} C_VEL
LIN {X 0,Y 559.911,Z 1071.004,A -85,B 0,C 180,E1 26186.417,E2 26186.417} C_VEL
LIN {X 0,Y 559.926,Z 1067.098,A -85,B 0,C 180,E1 26184.569,E2 26184.569} C_VEL
LIN {X 0,Y 559.956,Z 1061.469,A -85,B 0,C 180,E1 26182.717,E2 26182.717} C_VEL
LIN {X 0,Y 560.027,Z 1054.426,A -85,B 0,C 180,E1 26180.961,E2 26180.961} C_VEL
LIN {X 0,Y 560.142,Z 1045.515,A -85,B 0,C 180,E1 26179.198,E2 26179.198} C_VEL
LIN {X 0,Y 560.307,Z 1035.151,A -85,B 0,C 180,E1 26177.53,E2 26177.53} C_VEL
LIN {X 0,Y 560.531,Z 1023.35,A -85,B 0,C 180,E1 26175.961,E2 26175.961} C_VEL
LIN {X 0,Y 560.823,Z 1009.801,A -85,B 0,C 180,E1 26174.459,E2 26174.459} C_VEL
LIN {X 0,Y 561.16,Z 995.031,A -85,B 0,C 180,E1 26173.099,E2 26173.099} C_VEL
LIN {X 0,Y 561.528,Z 979.231,A -85,B 0,C 180,E1 26171.898,E2 26171.898} C_VEL
LIN {X 0,Y 561.872,Z 962.045,A -85,B 0,C 180,E1 26170.833,E2 26170.833} C_VEL
LIN {X 0,Y 562.257,Z 944.803,A -85,B 0,C 180,E1 26169.982,E2 26169.982} C_VEL
LIN {X 0,Y 562.557,Z 926.525,A -85,B 0,C 180,E1 26169.287,E2 26169.287} C_VEL
LIN {X 0,Y 562.813,Z 907.948,A -85,B 0,C 180,E1 26168.782,E2 26168.782} C_VEL
LIN {X 0,Y 562.978,Z 887.618,A -85,B 0,C 180,E1 26168.437,E2 26168.437} C_VEL
LIN {X 0,Y 563.549,Z 697.034,A -85,B 0,C 180,E1 26165.878,E2 26165.878} C_VEL
LIN {X 0,Y 562.754,Z 691.284,A -85,B 0,C 180,E1 26165.738,E2 26165.738} C_VEL
LIN {X 0,Y 563.496,Z 644.387,A -85,B 0,C 180,E1 26162.412,E2 26162.412} C_VEL
LIN {X 0,Y 564.382,Z 601.066,A -85,B 0,C 180,E1 26159.262,E2 26159.262} C_VEL
LIN {X 0,Y 564.386,Z 597.982,A -85,B 0,C 180,E1 26159.031,E2 26159.031} C_VEL
LIN {X 0,Y 560.284,Z 586.32,A -85,B 0,C 180,E1 26157.903,E2 26157.903} C_VEL
LIN {X 0,Y 560.267,Z 586.003,A -85,B 0,C 180,E1 26156.779,E2 26156.779} C_VEL
LIN {X 0,Y 560.224,Z 586.013,A -85,B 0,C 180,E1 26153.536,E2 26153.536} C_VEL
LIN {X 0,Y 560.287,Z 586.004,A -85,B 0,C 180,E1 26150.425,E2 26150.425} C_VEL
LIN {X 0,Y 560.217,Z 586.009,A -85,B 0,C 180,E1 26147.157,E2 26147.157} C_VEL
LIN {X 0,Y 560.286,Z 586.006,A -85,B 0,C 180,E1 26143.963,E2 26143.963} C_VEL
LIN {X 0,Y 560.217,Z 586.009,A -85,B 0,C 180,E1 26140.785,E2 26140.785} C_VEL
LIN {X 0,Y 560.284,Z 586.006,A -85,B 0,C 180,E1 26137.595,E2 26137.595} C_VEL
LIN {X 0,Y 560.223,Z 586.007,A -85,B 0,C 180,E1 26134.455,E2 26134.455} C_VEL
LIN {X 0,Y 560.274,Z 586.008,A -85,B 0,C 180,E1 26131.167,E2 26131.167} C_VEL
LIN {X 0,Y 560.237,Z 586.004,A -85,B 0,C 180,E1 26127.994,E2 26127.994} C_VEL
LIN {X 0,Y 560.234,Z 586.008,A -85,B 0,C 180,E1 26124.572,E2 26124.572} C_VEL
LIN {X 0,Y 560.266,Z 586.004,A -85,B 0,C 180,E1 26121.46,E2 26121.46} C_VEL
LIN {X 0,Y 560.228,Z 586.009,A -85,B 0,C 180,E1 26118.199,E2 26118.199} C_VEL
LIN {X 0,Y 560.284,Z 586.003,A -85,B 0,C 180,E1 26114.996,E2 26114.996} C_VEL
LIN {X 0,Y 560.227,Z 586.008,A -85,B 0,C 180,E1 26111.739,E2 26111.739} C_VEL
LIN {X 0,Y 560.283,Z 586.003,A -85,B 0,C 180,E1 26108.518,E2 26108.518} C_VEL
LIN {X 0,Y 560.231,Z 586.004,A -85,B 0,C 180,E1 26105.325,E2 26105.325} C_VEL
LIN {X 0,Y 560.272,Z 586.011,A -85,B 0,C 180,E1 26102.025,E2 26102.025} C_VEL
LIN {X 0,Y 560.25,Z 586.002,A -85,B 0,C 180,E1 26098.773,E2 26098.773} C_VEL
LIN {X 0,Y 560.244,Z 586.005,A -85,B 0,C 180,E1 26095.393,E2 26095.393} C_VEL
LIN {X 0,Y 560.28,Z 586.003,A -85,B 0,C 180,E1 26092.205,E2 26092.205} C_VEL
LIN {X 0,Y 560.238,Z 586.007,A -85,B 0,C 180,E1 26088.887,E2 26088.887} C_VEL
LIN {X 0,Y 560.28,Z 586.004,A -85,B 0,C 180,E1 26085.637,E2 26085.637} C_VEL
LIN {X 0,Y 560.241,Z 586.004,A -85,B 0,C 180,E1 26082.369,E2 26082.369} C_VEL
LIN {X 0,Y 560.283,Z 586.007,A -85,B 0,C 180,E1 26079.089,E2 26079.089} C_VEL
LIN {X 0,Y 560.241,Z 586.004,A -85,B 0,C 180,E1 26076.338,E2 26076.338} C_VEL
LIN {X 0,Y 559.256,Z 586.129,A -85,B 0,C 180,E1 26075.551,E2 26075.551} C_VEL
LIN {X 0,Y 552.875,Z 586.929,A -85,B 0,C 180,E1 26073.338,E2 26073.338} C_VEL
LIN {X 0,Y 552.339,Z 586.998,A -85,B 0,C 180,E1 26072.762,E2 26072.762} C_VEL
LIN {X 0,Y 552.332,Z 586.993,A -85,B 0,C 180,E1 26069.424,E2 26069.424} C_VEL
LIN {X 0,Y 552.311,Z 586.997,A -85,B 0,C 180,E1 26066.009,E2 26066.009} C_VEL
LIN {X 0,Y 552.339,Z 586.998,A -85,B 0,C 180,E1 26062.797,E2 26062.797} C_VEL
LIN {X 0,Y 552.311,Z 587.001,A -85,B 0,C 180,E1 26059.494,E2 26059.494} C_VEL
LIN {X 0,Y 552.381,Z 587.276,A -85,B 0,C 180,E1 26058.509,E2 26058.509} C_VEL
LIN {X 0,Y 554.925,Z 597.049,A -85,B 0,C 180,E1 26057.166,E2 26057.166} C_VEL
LIN {X 0,Y 554.122,Z 626.151,A -85,B 0,C 180,E1 26053.716,E2 26053.716} C_VEL
LIN {X 0,Y 553.531,Z 654.887,A -85,B 0,C 180,E1 26050.427,E2 26050.427} C_VEL
LIN {X 0,Y 553.05,Z 685.457,A -85,B 0,C 180,E1 26047.016,E2 26047.016} C_VEL
LIN {X 0,Y 552.764,Z 709.941,A -85,B 0,C 180,E1 26044.358,E2 26044.358} C_VEL
LIN {X 0,Y 553.458,Z 717.596,A -85,B 0,C 180,E1 26044.22,E2 26044.22} C_VEL
LIN {X 0,Y 553.148,Z 821.393,A -85,B 0,C 180,E1 26042.842,E2 26042.842} C_VEL
LIN {X 0,Y 553.042,Z 835.544,A -85,B 0,C 180,E1 26042.477,E2 26042.477} C_VEL
LIN {X 0,Y 552.861,Z 849.931,A -85,B 0,C 180,E1 26041.903,E2 26041.903} C_VEL
LIN {X 0,Y 552.654,Z 863.457,A -85,B 0,C 180,E1 26041.157,E2 26041.157} C_VEL
LIN {X 0,Y 552.44,Z 876.468,A -85,B 0,C 180,E1 26040.209,E2 26040.209} C_VEL
LIN {X 0,Y 552.263,Z 888.291,A -85,B 0,C 180,E1 26039.085,E2 26039.085} C_VEL
LIN {X 0,Y 552.122,Z 898.081,A -85,B 0,C 180,E1 26037.903,E2 26037.903} C_VEL
LIN {X 0,Y 552.021,Z 905.999,A -85,B 0,C 180,E1 26036.692,E2 26036.692} C_VEL
LIN {X 0,Y 551.958,Z 913.422,A -85,B 0,C 180,E1 26035.195,E2 26035.195} C_VEL
LIN {X 0,Y 551.928,Z 918.645,A -85,B 0,C 180,E1 26033.714,E2 26033.714} C_VEL
LIN {X 0,Y 551.919,Z 922.082,A -85,B 0,C 180,E1 26032.22,E2 26032.22} C_VEL
LIN {X 0,Y 551.917,Z 923.854,A -85,B 0,C 180,E1 26030.576,E2 26030.576} C_VEL
LIN {X 0,Y 551.918,Z 923.623,A -85,B 0,C 180,E1 26028.974,E2 26028.974} C_VEL
LIN {X 0,Y 551.919,Z 921.74,A -85,B 0,C 180,E1 26027.501,E2 26027.501} C_VEL
LIN {X 0,Y 551.93,Z 918.024,A -85,B 0,C 180,E1 26025.983,E2 26025.983} C_VEL
LIN {X 0,Y 551.962,Z 912.842,A -85,B 0,C 180,E1 26024.584,E2 26024.584} C_VEL
LIN {X 0,Y 552.022,Z 905.851,A -85,B 0,C 180,E1 26023.192,E2 26023.192} C_VEL
LIN {X 0,Y 552.141,Z 896.605,A -85,B 0,C 180,E1 26021.808,E2 26021.808} C_VEL
LIN {X 0,Y 552.296,Z 886.559,A -85,B 0,C 180,E1 26020.641,E2 26020.641} C_VEL
LIN {X 0,Y 552.459,Z 875.028,A -85,B 0,C 180,E1 26019.585,E2 26019.585} C_VEL
LIN {X 0,Y 552.669,Z 862.446,A -85,B 0,C 180,E1 26018.688,E2 26018.688} C_VEL
LIN {X 0,Y 552.878,Z 848.747,A -85,B 0,C 180,E1 26017.952,E2 26017.952} C_VEL
LIN {X 0,Y 553.049,Z 834.585,A -85,B 0,C 180,E1 26017.404,E2 26017.404} C_VEL
LIN {X 0,Y 553.171,Z 819.158,A -85,B 0,C 180,E1 26017.024,E2 26017.024} C_VEL
LIN {X 0,Y 553.243,Z 713.678,A -85,B 0,C 180,E1 26015.633,E2 26015.633} C_VEL
LIN {X 0,Y 552.746,Z 709.543,A -85,B 0,C 180,E1 26015.527,E2 26015.527} C_VEL
LIN {X 0,Y 553.147,Z 678.037,A -85,B 0,C 180,E1 26012.072,E2 26012.072} C_VEL
LIN {X 0,Y 553.649,Z 647.546,A -85,B 0,C 180,E1 26008.655,E2 26008.655} C_VEL
LIN {X 0,Y 554.258,Z 618.779,A -85,B 0,C 180,E1 26005.343,E2 26005.343} C_VEL
LIN {X 0,Y 554.843,Z 596.82,A -85,B 0,C 180,E1 26002.753,E2 26002.753} C_VEL
LIN {X 0,Y 552.346,Z 587.101,A -85,B 0,C 180,E1 26001.385,E2 26001.385} C_VEL
LIN {X 0,Y 552.323,Z 586.997,A -85,B 0,C 180,E1 25998.09,E2 25998.09} C_VEL
LIN {X 0,Y 552.33,Z 586.994,A -85,B 0,C 180,E1 25994.769,E2 25994.769} C_VEL
LIN {X 0,Y 552.329,Z 586.997,A -85,B 0,C 180,E1 25991.421,E2 25991.421} C_VEL
LIN {X 0,Y 552.332,Z 586.991,A -85,B 0,C 180,E1 25987.95,E2 25987.95} C_VEL
LIN {X 0,Y 552.336,Z 586.996,A -85,B 0,C 180,E1 25984.594,E2 25984.594} C_VEL
LIN {X 0,Y 552.317,Z 586.994,A -85,B 0,C 180,E1 25981.332,E2 25981.332} C_VEL
LIN {X 0,Y 552.333,Z 586.987,A -85,B 0,C 180,E1 25978.089,E2 25978.089} C_VEL
LIN {X 0,Y 552.323,Z 586.998,A -85,B 0,C 180,E1 25974.73,E2 25974.73} C_VEL
LIN {X 0,Y 552.328,Z 586.99,A -85,B 0,C 180,E1 25971.282,E2 25971.282} C_VEL
LIN {X 0,Y 552.338,Z 586.991,A -85,B 0,C 180,E1 25967.919,E2 25967.919} C_VEL
LIN {X 0,Y 552.311,Z 586.994,A -85,B 0,C 180,E1 25964.621,E2 25964.621} C_VEL
LIN {X 0,Y 552.339,Z 586.984,A -85,B 0,C 180,E1 25961.301,E2 25961.301} C_VEL
LIN {X 0,Y 552.32,Z 586.997,A -85,B 0,C 180,E1 25957.989,E2 25957.989} C_VEL
LIN {X 0,Y 552.317,Z 586.987,A -85,B 0,C 180,E1 25954.515,E2 25954.515} C_VEL
LIN {X 0,Y 552.338,Z 586.995,A -85,B 0,C 180,E1 25951.18,E2 25951.18} C_VEL
LIN {X 0,Y 552.305,Z 586.994,A -85,B 0,C 180,E1 25947.938,E2 25947.938} C_VEL
LIN {X 0,Y 552.342,Z 586.988,A -85,B 0,C 180,E1 25944.605,E2 25944.605} C_VEL
LIN {X 0,Y 552.311,Z 586.999,A -85,B 0,C 180,E1 25941.339,E2 25941.339} C_VEL
LIN {X 0,Y 552.317,Z 586.984,A -85,B 0,C 180,E1 25937.924,E2 25937.924} C_VEL
LIN {X 0,Y 552.346,Z 586.996,A -85,B 0,C 180,E1 25934.574,E2 25934.574} C_VEL
LIN {X 0,Y 552.299,Z 586.994,A -85,B 0,C 180,E1 25931.275,E2 25931.275} C_VEL
LIN {X 0,Y 552.343,Z 586.987,A -85,B 0,C 180,E1 25928.013,E2 25928.013} C_VEL
LIN {X 0,Y 552.3,Z 586.997,A -85,B 0,C 180,E1 25924.777,E2 25924.777} C_VEL
LIN {X 0,Y 552.33,Z 586.984,A -85,B 0,C 180,E1 25921.452,E2 25921.452} C_VEL
LIN {X 0,Y 552.33,Z 586.997,A -85,B 0,C 180,E1 25918.133,E2 25918.133} C_VEL
LIN {X 0,Y 552.298,Z 586.993,A -85,B 0,C 180,E1 25914.807,E2 25914.807} C_VEL
LIN {X 0,Y 552.346,Z 586.993,A -85,B 0,C 180,E1 25911.569,E2 25911.569} C_VEL
LIN {X 0,Y 552.289,Z 586.997,A -85,B 0,C 180,E1 25908.302,E2 25908.302} C_VEL
LIN {X 0,Y 552.345,Z 586.988,A -85,B 0,C 180,E1 25904.998,E2 25904.998} C_VEL
LIN {X 0,Y 552.3,Z 586.999,A -85,B 0,C 180,E1 25901.748,E2 25901.748} C_VEL
LIN {X 0,Y 552.305,Z 586.991,A -85,B 0,C 180,E1 25898.327,E2 25898.327} C_VEL
LIN {X 0,Y 552.342,Z 586.995,A -85,B 0,C 180,E1 25895.053,E2 25895.053} C_VEL
LIN {X 0,Y 552.286,Z 586.997,A -85,B 0,C 180,E1 25891.803,E2 25891.803} C_VEL
LIN {X 0,Y 552.348,Z 586.994,A -85,B 0,C 180,E1 25888.578,E2 25888.578} C_VEL
LIN {X 0,Y 552.28,Z 586.997,A -85,B 0,C 180,E1 25885.356,E2 25885.356} C_VEL
LIN {X 0,Y 552.346,Z 586.99,A -85,B 0,C 180,E1 25882.116,E2 25882.116} C_VEL
LIN {X 0,Y 552.29,Z 587,A -85,B 0,C 180,E1 25878.916,E2 25878.916} C_VEL
LIN {X 0,Y 552.31,Z 586.993,A -85,B 0,C 180,E1 25875.525,E2 25875.525} C_VEL
LIN {X 0,Y 552.32,Z 586.999,A -85,B 0,C 180,E1 25872.333,E2 25872.333} C_VEL
LIN {X 0,Y 552.288,Z 586.997,A -85,B 0,C 180,E1 25869.044,E2 25869.044} C_VEL
LIN {X 0,Y 552.336,Z 587,A -85,B 0,C 180,E1 25865.911,E2 25865.911} C_VEL
LIN {X 0,Y 552.283,Z 587.017,A -85,B 0,C 180,E1 25862.65,E2 25862.65} C_VEL
LIN {X 0,Y 552.371,Z 587.555,A -85,B 0,C 180,E1 25862.46,E2 25862.46} C_VEL
LIN {X 0,Y 557.079,Z 601.404,A -85,B 0,C 180,E1 25861.115,E2 25861.115} C_VEL
LIN {X 0,Y 556.275,Z 639.655,A -85,B 0,C 180,E1 25858.328,E2 25858.328} C_VEL
LIN {X 0,Y 555.422,Z 682.976,A -85,B 0,C 180,E1 25855.198,E2 25855.198} C_VEL
LIN {X 0,Y 555.358,Z 692.228,A -85,B 0,C 180,E1 25854.571,E2 25854.571} C_VEL
LIN {X 0,Y 556.397,Z 700.968,A -85,B 0,C 180,E1 25854.397,E2 25854.397} C_VEL
LIN {X 0,Y 555.438,Z 901.304,A -85,B 0,C 180,E1 25851.656,E2 25851.656} C_VEL
LIN {X 0,Y 555.161,Z 920.272,A -85,B 0,C 180,E1 25851.202,E2 25851.202} C_VEL
LIN {X 0,Y 554.834,Z 938.392,A -85,B 0,C 180,E1 25850.574,E2 25850.574} C_VEL
LIN {X 0,Y 554.413,Z 956.039,A -85,B 0,C 180,E1 25849.764,E2 25849.764} C_VEL
LIN {X 0,Y 553.991,Z 972.794,A -85,B 0,C 180,E1 25848.792,E2 25848.792} C_VEL
LIN {X 0,Y 553.575,Z 988.625,A -85,B 0,C 180,E1 25847.665,E2 25847.665} C_VEL
LIN {X 0,Y 553.164,Z 1003.554,A -85,B 0,C 180,E1 25846.378,E2 25846.378} C_VEL
LIN {X 0,Y 552.809,Z 1017.017,A -85,B 0,C 180,E1 25844.99,E2 25844.99} C_VEL
LIN {X 0,Y 552.498,Z 1029.911,A -85,B 0,C 180,E1 25843.394,E2 25843.394} C_VEL
LIN {X 0,Y 552.263,Z 1041.229,A -85,B 0,C 180,E1 25841.699,E2 25841.699} C_VEL
LIN {X 0,Y 552.095,Z 1051.173,A -85,B 0,C 180,E1 25839.87,E2 25839.87} C_VEL
LIN {X 0,Y 551.988,Z 1059.177,A -85,B 0,C 180,E1 25838.018,E2 25838.018} C_VEL
LIN {X 0,Y 551.942,Z 1065.411,A -85,B 0,C 180,E1 25836.136,E2 25836.136} C_VEL
LIN {X 0,Y 551.922,Z 1069.876,A -85,B 0,C 180,E1 25834.26,E2 25834.26} C_VEL
LIN {X 0,Y 551.915,Z 1072.792,A -85,B 0,C 180,E1 25832.284,E2 25832.284} C_VEL
LIN {X 0,Y 551.908,Z 1073.94,A -85,B 0,C 180,E1 25830.312,E2 25830.312} C_VEL
LIN {X 0,Y 551.913,Z 1073.348,A -85,B 0,C 180,E1 25828.339,E2 25828.339} C_VEL
LIN {X 0,Y 551.912,Z 1071.004,A -85,B 0,C 180,E1 25826.365,E2 25826.365} C_VEL
LIN {X 0,Y 551.928,Z 1067.098,A -85,B 0,C 180,E1 25824.491,E2 25824.491} C_VEL
LIN {X 0,Y 551.967,Z 1061.469,A -85,B 0,C 180,E1 25822.611,E2 25822.611} C_VEL
LIN {X 0,Y 552.054,Z 1054.214,A -85,B 0,C 180,E1 25820.781,E2 25820.781} C_VEL
LIN {X 0,Y 552.187,Z 1045.516,A -85,B 0,C 180,E1 25819.04,E2 25819.04} C_VEL
LIN {X 0,Y 552.389,Z 1034.981,A -85,B 0,C 180,E1 25817.323,E2 25817.323} C_VEL
LIN {X 0,Y 552.654,Z 1023.35,A -85,B 0,C 180,E1 25815.756,E2 25815.756} C_VEL
LIN {X 0,Y 553.007,Z 1009.576,A -85,B 0,C 180,E1 25814.21,E2 25814.21} C_VEL
LIN {X 0,Y 553.415,Z 994.603,A -85,B 0,C 180,E1 25812.819,E2 25812.819} C_VEL
LIN {X 0,Y 553.853,Z 978.432,A -85,B 0,C 180,E1 25811.584,E2 25811.584} C_VEL
LIN {X 0,Y 554.246,Z 962.047,A -85,B 0,C 180,E1 25810.559,E2 25810.559} C_VEL
LIN {X 0,Y 554.692,Z 944.805,A -85,B 0,C 180,E1 25809.697,E2 25809.697} C_VEL
LIN {X 0,Y 555.046,Z 926.528,A -85,B 0,C 180,E1 25808.993,E2 25808.993} C_VEL
LIN {X 0,Y 555.347,Z 907.92,A -85,B 0,C 180,E1 25808.482,E2 25808.482} C_VEL
LIN {X 0,Y 555.539,Z 887.491,A -85,B 0,C 180,E1 25808.132,E2 25808.132} C_VEL
LIN {X 0,Y 556.243,Z 698.106,A -85,B 0,C 180,E1 25805.556,E2 25805.556} C_VEL
LIN {X 0,Y 555.291,Z 691.622,A -85,B 0,C 180,E1 25805.409,E2 25805.409} C_VEL
LIN {X 0,Y 556.142,Z 645.963,A -85,B 0,C 180,E1 25802.132,E2 25802.132} C_VEL
LIN {X 0,Y 556.997,Z 606.145,A -85,B 0,C 180,E1 25799.23,E2 25799.23} C_VEL
LIN {X 0,Y 556.961,Z 600.548,A -85,B 0,C 180,E1 25798.815,E2 25798.815} C_VEL
LIN {X 0,Y 552.325,Z 587.315,A -85,B 0,C 180,E1 25797.507,E2 25797.507} C_VEL
LIN {X 0,Y 552.344,Z 586.992,A -85,B 0,C 180,E1 25796.564,E2 25796.564} C_VEL
LIN {X 0,Y 552.279,Z 587.002,A -85,B 0,C 180,E1 25793.323,E2 25793.323} C_VEL
LIN {X 0,Y 552.347,Z 586.996,A -85,B 0,C 180,E1 25790.132,E2 25790.132} C_VEL
LIN {X 0,Y 552.28,Z 586.997,A -85,B 0,C 180,E1 25786.958,E2 25786.958} C_VEL
LIN {X 0,Y 552.342,Z 586.997,A -85,B 0,C 180,E1 25783.749,E2 25783.749} C_VEL
LIN {X 0,Y 552.294,Z 586.996,A -85,B 0,C 180,E1 25780.504,E2 25780.504} C_VEL
LIN {X 0,Y 552.295,Z 587,A -85,B 0,C 180,E1 25777.074,E2 25777.074} C_VEL
LIN {X 0,Y 552.332,Z 586.992,A -85,B 0,C 180,E1 25773.887,E2 25773.887} C_VEL
LIN {X 0,Y 552.282,Z 586.999,A -85,B 0,C 180,E1 25770.579,E2 25770.579} C_VEL
LIN {X 0,Y 552.346,Z 586.992,A -85,B 0,C 180,E1 25767.374,E2 25767.374} C_VEL
LIN {X 0,Y 552.284,Z 586.994,A -85,B 0,C 180,E1 25764.151,E2 25764.151} C_VEL
LIN {X 0,Y 552.343,Z 586.999,A -85,B 0,C 180,E1 25760.892,E2 25760.892} C_VEL
LIN {X 0,Y 552.293,Z 586.995,A -85,B 0,C 180,E1 25757.706,E2 25757.706} C_VEL
LIN {X 0,Y 552.314,Z 586.997,A -85,B 0,C 180,E1 25754.36,E2 25754.36} C_VEL
LIN {X 0,Y 552.32,Z 586.993,A -85,B 0,C 180,E1 25751.134,E2 25751.134} C_VEL
LIN {X 0,Y 552.297,Z 586.998,A -85,B 0,C 180,E1 25747.803,E2 25747.803} C_VEL
LIN {X 0,Y 552.342,Z 586.99,A -85,B 0,C 180,E1 25744.568,E2 25744.568} C_VEL
LIN {X 0,Y 552.292,Z 586.995,A -85,B 0,C 180,E1 25741.245,E2 25741.245} C_VEL
LIN {X 0,Y 552.339,Z 586.998,A -85,B 0,C 180,E1 25737.925,E2 25737.925} C_VEL
LIN {X 0,Y 552.313,Z 586.989,A -85,B 0,C 180,E1 25734.598,E2 25734.598} C_VEL
LIN {X 0,Y 552.304,Z 586.992,A -85,B 0,C 180,E1 25731.148,E2 25731.148} C_VEL
LIN {X 0,Y 552.341,Z 586.994,A -85,B 0,C 180,E1 25727.878,E2 25727.878} C_VEL
LIN {X 0,Y 552.299,Z 586.996,A -85,B 0,C 180,E1 25724.566,E2 25724.566} C_VEL
LIN {X 0,Y 552.341,Z 586.999,A -85,B 0,C 180,E1 25721.218,E2 25721.218} C_VEL
LIN {X 0,Y 552.322,Z 586.993,A -85,B 0,C 180,E1 25717.88,E2 25717.88} C_VEL
LIN {X 0,Y 552.313,Z 586.997,A -85,B 0,C 180,E1 25714.478,E2 25714.478} C_VEL
